	{attribute 'c++_compatible'}
	{attribute 'external_name' := 'FB_VN_ReadRegister_UDINT_GUID_B1D0CDA5_1E02_2B99_6D2D_309CAE674913'}
	{attribute 'TcIecLibraryType'}
	(* This FB reads a DINT register from the camera. Requires an open control channel (e.g. by calling FB_VN_GevCameraControl.OpenCamera() before) *)
	FUNCTION_BLOCK FB_VN_ReadRegister_UDINT
	VAR_INPUT
		(* The address of the register that should be read *)
		 {attribute 'GUID' := 'E1ED2436-3512-43FA-B927-3F71DEDDA853'}
		nAddress : GVCP_REGISTER_ADDRESS;
		(* OPTIONAL: The endianness of the register. 0 = Big, 1 = Little. Default: 0 *)
		nEndian : UINT;
		(* Reading the register is triggered by a rising edge at this input. *)
		bRead : BOOL;
	END_VAR
	VAR
		 {attribute 'hide'}
		_reserved1 : USINT;
	END_VAR
	VAR_INPUT
		(* Indicates the time before the function is cancelled. *)
		nTimeout : TIME := VISION_ADS_TIMEOUT;
	END_VAR
	VAR_OUTPUT
		(* The read value *)
		nValue : UDINT;
		(* This output remains TRUE until the function block has executed a command, but at the longest for the duration supplied to the 'nTimeout' input. While bBusy = TRUE, no new command will be accepted at the inputs. *)
		bBusy : BOOL;
		(* This output is switched to TRUE as soon as an error occurs during the execution of a command. The command-specific error code is contained in ‘nErrorId’. If the function block has a timeout error, 'bError' is TRUE and 'nErrorId' is 1861 (hexadecimal 0x745). Is reset to FALSE by the execution of a command at the inputs. *)
		bError : BOOL;
	END_VAR
	VAR
		 {attribute 'hide'}
		_reserved2 : UINT;
	END_VAR
	VAR_OUTPUT
		(* Contains the ADS error code or the command-specific error code of the last executed command. Is reset to 0 by the execution of a command at the inputs. *)
		nErrorId : UDINT;
	END_VAR
	VAR
		(* Internal reference to the corresponding TcVnGevImageProvider TcCOM module ID, which needs to be set via TC init symbol. *)
		{attribute 'TcInitSymbol'}
		{attribute 'TcCategoryOID' := 'TcVnGevImageProvider'}
		 {attribute 'GUID' := '18071995-0000-0000-0000-00000000000F'}
		oidITcVnGevImageProvider : OTCID;
		 {attribute 'hide'}
		_reserved3 : UINT_0_32;
		(* Internal reference to the corresponding TcVnGevImageProvider module. *)
		{attribute 'hide'}
		 {attribute 'GUID' := 'ED7659DB-95DC-4A4A-B62F-02C9870D5E81'}
		ipGevImageProvider : ITcVnGevImageProvider;
		(* Internal timestamp for timeout detection *)
		{attribute 'hide'}
		nTimeElapsed : TIME;
		(* Internal flag for rising edge detection *)
		{attribute 'hide'}
		bLastRead : BOOL;
		 {attribute 'hide'}
		_reserved4 : ARRAY [1..3] OF USINT;
	END_VAR


	(* Internal method *)
	{attribute 'hide'}
	METHOD FB_exit : BOOL
	VAR_INPUT
		(*  if TRUE, the exit method is called for exiting an instance that is copied afterwards (online change). *)
		bInCopyCode : BOOL;
	END_VAR
END_METHOD


	(* Internal method *)
	{attribute 'hide'}
	METHOD FB_init : BOOL
	VAR_INPUT
		(*  if TRUE, the retain variables are initialized (warm start / cold start) *)
		bInitRetains : BOOL;
		(*  if TRUE, the instance afterwards gets moved into the copy code (online change) *)
		bInCopyCode : BOOL;
	END_VAR
END_METHOD

END_FUNCTION_BLOCK

// Function Blocks/Camera Register Access/FB_VN_WriteRegister_UDINT

	{attribute 'c++_compatible'}
	{attribute 'external_name' := 'FB_VN_WriteRegister_UDINT_GUID_AF8CFF3D_C541_213B_73EF_5E560CA3A7B1'}
	{attribute 'TcIecLibraryType'}
	(* This FB writes a DINT value into a register on the camera. Requires an open control channel (e.g. by calling FB_VN_GevCameraControl.OpenCamera() before) *)
	FUNCTION_BLOCK FB_VN_WriteRegister_UDINT
	VAR_INPUT
		(* The address of the register that should be written *)
		 {attribute 'GUID' := 'E1ED2436-3512-43FA-B927-3F71DEDDA853'}
		nAddress : GVCP_REGISTER_ADDRESS;
		(* The value to write *)
		nValue : UDINT;
		(* OPTIONAL: The endianness of the register. 0 = Big, 1 = Little. Default: 0 *)
		nEndian : UINT;
		(* Writing the register is triggered by a rising edge at this input. *)
		bWrite : BOOL;
	END_VAR
	VAR
		 {attribute 'hide'}
		_reserved1 : USINT;
	END_VAR
	VAR_INPUT
		(* Indicates the time before the function is cancelled. *)
		nTimeout : TIME := VISION_ADS_TIMEOUT;
	END_VAR
	VAR_OUTPUT
		(* This output remains TRUE until the function block has executed a command, but at the longest for the duration supplied to the 'nTimeout' input. While bBusy = TRUE, no new command will be accepted at the inputs. *)
		bBusy : BOOL;
		(* This output is switched to TRUE as soon as an error occurs during the execution of a command. The command-specific error code is contained in ‘nErrorId’. If the function block has a timeout error, 'bError' is TRUE and 'nErrorId' is 1861 (hexadecimal 0x745). Is reset to FALSE by the execution of a command at the inputs. *)
		bError : BOOL;
	END_VAR
	VAR
		 {attribute 'hide'}
		_reserved2 : UINT;
	END_VAR
	VAR_OUTPUT
		(* Contains the ADS error code or the command-specific error code of the last executed command. Is reset to 0 by the execution of a command at the inputs. *)
		nErrorId : UDINT;
	END_VAR
	VAR
		(* Internal reference to the corresponding TcVnGevImageProvider TcCOM module ID, which needs to be set via TC init symbol. *)
		{attribute 'TcInitSymbol'}
		{attribute 'TcCategoryOID' := 'TcVnGevImageProvider'}
		 {attribute 'GUID' := '18071995-0000-0000-0000-00000000000F'}
		oidITcVnGevImageProvider : OTCID;
		 {attribute 'hide'}
		_reserved3 : UINT_0_32;
		(* Internal reference to the corresponding TcVnGevImageProvider module. *)
		{attribute 'hide'}
		 {attribute 'GUID' := 'ED7659DB-95DC-4A4A-B62F-02C9870D5E81'}
		ipGevImageProvider : ITcVnGevImageProvider;
		(* Internal timestamp for timeout detection *)
		{attribute 'hide'}
		nTimeElapsed : TIME;
		(* Internal flag for rising edge detection *)
		{attribute 'hide'}
		bLastWrite : BOOL;
		 {attribute 'hide'}
		_reserved4 : ARRAY [1..3] OF USINT;
	END_VAR


	(* Internal method *)
	{attribute 'hide'}
	METHOD FB_exit : BOOL
	VAR_INPUT
		(*  if TRUE, the exit method is called for exiting an instance that is copied afterwards (online change). *)
		bInCopyCode : BOOL;
	END_VAR
END_METHOD


	(* Internal method *)
	{attribute 'hide'}
	METHOD FB_init : BOOL
	VAR_INPUT
		(*  if TRUE, the retain variables are initialized (warm start / cold start) *)
		bInitRetains : BOOL;
		(*  if TRUE, the instance afterwards gets moved into the copy code (online change) *)
		bInCopyCode : BOOL;
	END_VAR
END_METHOD

END_FUNCTION_BLOCK

// Function Blocks/Camera Register Access/FB_VN_ReadRegister_ULINT

	{attribute 'c++_compatible'}
	{attribute 'external_name' := 'FB_VN_ReadRegister_ULINT_GUID_6D8277AF_24E6_2571_66A8_DA51E0B530F6'}
	{attribute 'TcIecLibraryType'}
	(* This FB reads a ULINT register from the camera. Requires an open control channel (e.g. by calling FB_VN_GevCameraControl.OpenCamera() before) *)
	FUNCTION_BLOCK FB_VN_ReadRegister_ULINT
	VAR_INPUT
		(* The address of the register that should be read *)
		 {attribute 'GUID' := 'E1ED2436-3512-43FA-B927-3F71DEDDA853'}
		nAddress : GVCP_REGISTER_ADDRESS;
		(* OPTIONAL: The endianness of the register. 0 = Big, 1 = Little. Default: 0 *)
		nEndian : UINT;
		(* Reading the register is triggered by a rising edge at this input. *)
		bRead : BOOL;
	END_VAR
	VAR
		 {attribute 'hide'}
		_reserved1 : USINT;
	END_VAR
	VAR_INPUT
		(* Indicates the time before the function is cancelled. *)
		nTimeout : TIME := VISION_ADS_TIMEOUT;
	END_VAR
	VAR
		 {attribute 'hide'}
		_reserved2 : UINT_0_32;
	END_VAR
	VAR_OUTPUT
		(* The read value *)
		nValue : ULINT;
		(* This output remains TRUE until the function block has executed a command, but at the longest for the duration supplied to the 'nTimeout' input. While bBusy = TRUE, no new command will be accepted at the inputs. *)
		bBusy : BOOL;
		(* This output is switched to TRUE as soon as an error occurs during the execution of a command. The command-specific error code is contained in ‘nErrorId’. If the function block has a timeout error, 'bError' is TRUE and 'nErrorId' is 1861 (hexadecimal 0x745). Is reset to FALSE by the execution of a command at the inputs. *)
		bError : BOOL;
	END_VAR
	VAR
		 {attribute 'hide'}
		_reserved3 : UINT;
	END_VAR
	VAR_OUTPUT
		(* Contains the ADS error code or the command-specific error code of the last executed command. Is reset to 0 by the execution of a command at the inputs. *)
		nErrorId : UDINT;
	END_VAR
	VAR
		(* Internal reference to the corresponding TcVnGevImageProvider TcCOM module ID, which needs to be set via TC init symbol. *)
		{attribute 'TcInitSymbol'}
		{attribute 'TcCategoryOID' := 'TcVnGevImageProvider'}
		 {attribute 'GUID' := '18071995-0000-0000-0000-00000000000F'}
		oidITcVnGevImageProvider : OTCID;
		 {attribute 'hide'}
		_reserved4 : UINT_0_32;
		(* Internal reference to the corresponding TcVnGevImageProvider module. *)
		{attribute 'hide'}
		 {attribute 'GUID' := 'ED7659DB-95DC-4A4A-B62F-02C9870D5E81'}
		ipGevImageProvider : ITcVnGevImageProvider;
		(* Internal timestamp for timeout detection *)
		{attribute 'hide'}
		nTimeElapsed : TIME;
		(* Internal flag for rising edge detection *)
		{attribute 'hide'}
		bLastRead : BOOL;
		 {attribute 'hide'}
		_reserved5 : ARRAY [1..3] OF USINT;
	END_VAR


	(* Internal method *)
	{attribute 'hide'}
	METHOD FB_exit : BOOL
	VAR_INPUT
		(*  if TRUE, the exit method is called for exiting an instance that is copied afterwards (online change). *)
		bInCopyCode : BOOL;
	END_VAR
END_METHOD


	(* Internal method *)
	{attribute 'hide'}
	METHOD FB_init : BOOL
	VAR_INPUT
		(*  if TRUE, the retain variables are initialized (warm start / cold start) *)
		bInitRetains : BOOL;
		(*  if TRUE, the instance afterwards gets moved into the copy code (online change) *)
		bInCopyCode : BOOL;
	END_VAR
END_METHOD

END_FUNCTION_BLOCK

// Function Blocks/Camera Register Access/FB_VN_WriteRegister_ULINT

	{attribute 'c++_compatible'}
	{attribute 'external_name' := 'FB_VN_WriteRegister_ULINT_GUID_F5D47CB9_E51C_2962_4F84_AA60BB261FC0'}
	{attribute 'TcIecLibraryType'}
	(* This FB writes a ULINT value into a register on the camera. Requires an open control channel (e.g. by calling FB_VN_GevCameraControl.OpenCamera() before) *)
	FUNCTION_BLOCK FB_VN_WriteRegister_ULINT
	VAR_INPUT
		(* The address of the register that should be written *)
		 {attribute 'GUID' := 'E1ED2436-3512-43FA-B927-3F71DEDDA853'}
		nAddress : GVCP_REGISTER_ADDRESS;
	END_VAR
	VAR
		 {attribute 'hide'}
		_reserved1 : UINT_0_32;
	END_VAR
	VAR_INPUT
		(* The value to write *)
		nValue : ULINT;
		(* OPTIONAL: The endianness of the register. 0 = Big, 1 = Little. Default: 0 *)
		nEndian : UINT;
		(* Writing the register is triggered by a rising edge at this input. *)
		bWrite : BOOL;
	END_VAR
	VAR
		 {attribute 'hide'}
		_reserved2 : USINT;
	END_VAR
	VAR_INPUT
		(* Indicates the time before the function is cancelled. *)
		nTimeout : TIME := VISION_ADS_TIMEOUT;
	END_VAR
	VAR_OUTPUT
		(* This output remains TRUE until the function block has executed a command, but at the longest for the duration supplied to the 'nTimeout' input. While bBusy = TRUE, no new command will be accepted at the inputs. *)
		bBusy : BOOL;
		(* This output is switched to TRUE as soon as an error occurs during the execution of a command. The command-specific error code is contained in ‘nErrorId’. If the function block has a timeout error, 'bError' is TRUE and 'nErrorId' is 1861 (hexadecimal 0x745). Is reset to FALSE by the execution of a command at the inputs. *)
		bError : BOOL;
	END_VAR
	VAR
		 {attribute 'hide'}
		_reserved3 : UINT;
	END_VAR
	VAR_OUTPUT
		(* Contains the ADS error code or the command-specific error code of the last executed command. Is reset to 0 by the execution of a command at the inputs. *)
		nErrorId : UDINT;
	END_VAR
	VAR
		(* Internal reference to the corresponding TcVnGevImageProvider TcCOM module ID, which needs to be set via TC init symbol. *)
		{attribute 'TcInitSymbol'}
		{attribute 'TcCategoryOID' := 'TcVnGevImageProvider'}
		 {attribute 'GUID' := '18071995-0000-0000-0000-00000000000F'}
		oidITcVnGevImageProvider : OTCID;
		 {attribute 'hide'}
		_reserved4 : UINT_0_32;
		(* Internal reference to the corresponding TcVnGevImageProvider module. *)
		{attribute 'hide'}
		 {attribute 'GUID' := 'ED7659DB-95DC-4A4A-B62F-02C9870D5E81'}
		ipGevImageProvider : ITcVnGevImageProvider;
		(* Internal timestamp for timeout detection *)
		{attribute 'hide'}
		nTimeElapsed : TIME;
		(* Internal flag for rising edge detection *)
		{attribute 'hide'}
		bLastWrite : BOOL;
		 {attribute 'hide'}
		_reserved5 : ARRAY [1..3] OF USINT;
	END_VAR


	(* Internal method *)
	{attribute 'hide'}
	METHOD FB_exit : BOOL
	VAR_INPUT
		(*  if TRUE, the exit method is called for exiting an instance that is copied afterwards (online change). *)
		bInCopyCode : BOOL;
	END_VAR
END_METHOD


	(* Internal method *)
	{attribute 'hide'}
	METHOD FB_init : BOOL
	VAR_INPUT
		(*  if TRUE, the retain variables are initialized (warm start / cold start) *)
		bInitRetains : BOOL;
		(*  if TRUE, the instance afterwards gets moved into the copy code (online change) *)
		bInCopyCode : BOOL;
	END_VAR
END_METHOD

END_FUNCTION_BLOCK

// Function Blocks/Camera Register Access/FB_VN_ReadMemory

	{attribute 'c++_compatible'}
	{attribute 'external_name' := 'FB_VN_ReadMemory_GUID_9CA954A7_F2A2_273A_543E_66E465761E40'}
	{attribute 'TcIecLibraryType'}
	(* This FB reads consecutive memory locations from the camera. Requires an open control channel (e.g. by calling FB_VN_GevCameraControl.OpenCamera() before) *)
	FUNCTION_BLOCK FB_VN_ReadMemory
	VAR_INPUT
		(* The address of the first byte to read from the camera (must be 32-bit aligned) *)
		 {attribute 'GUID' := 'E1ED2436-3512-43FA-B927-3F71DEDDA853'}
		nAddress : GVCP_REGISTER_ADDRESS;
		(* The number of bytes to read, starting with nAddress (must be a multiple of 4, not more than 536) *)
		nLength : UINT;
	END_VAR
	VAR
		 {attribute 'hide'}
		_reserved1 : UINT;
	END_VAR
	VAR_INPUT
		(* Pointer to the buffer where the read memory content is written to (The buffer must have a size of at least nLength bytes!) *)
		 {attribute 'GUID' := '18071995-0000-0000-0000-000000000018'}
		pBuffer : PVOID;
		(* Reading the memory is triggered by a rising edge at this input. *)
		bRead : BOOL;
	END_VAR
	VAR
		 {attribute 'hide'}
		_reserved2 : ARRAY [1..3] OF USINT;
	END_VAR
	VAR_INPUT
		(* Indicates the time before the function is cancelled. *)
		nTimeout : TIME := VISION_ADS_TIMEOUT;
	END_VAR
	VAR_OUTPUT
		(* This output remains TRUE until the function block has executed a command, but at the longest for the duration supplied to the 'nTimeout' input. While bBusy = TRUE, no new command will be accepted at the inputs. *)
		bBusy : BOOL;
		(* This output is switched to TRUE as soon as an error occurs during the execution of a command. The command-specific error code is contained in ‘nErrorId’. If the function block has a timeout error, 'bError' is TRUE and 'nErrorId' is 1861 (hexadecimal 0x745). Is reset to FALSE by the execution of a command at the inputs. *)
		bError : BOOL;
	END_VAR
	VAR
		 {attribute 'hide'}
		_reserved3 : UINT;
	END_VAR
	VAR_OUTPUT
		(* Contains the ADS error code or the command-specific error code of the last executed command. Is reset to 0 by the execution of a command at the inputs. *)
		nErrorId : UDINT;
	END_VAR
	VAR
		(* Internal reference to the corresponding TcVnGevImageProvider TcCOM module ID, which needs to be set via TC init symbol. *)
		{attribute 'TcInitSymbol'}
		{attribute 'TcCategoryOID' := 'TcVnGevImageProvider'}
		 {attribute 'GUID' := '18071995-0000-0000-0000-00000000000F'}
		oidITcVnGevImageProvider : OTCID;
		 {attribute 'hide'}
		_reserved4 : UINT_0_32;
		(* Internal reference to the corresponding TcVnGevImageProvider module. *)
		{attribute 'hide'}
		 {attribute 'GUID' := 'ED7659DB-95DC-4A4A-B62F-02C9870D5E81'}
		ipGevImageProvider : ITcVnGevImageProvider;
		(* Internal timestamp for timeout detection *)
		{attribute 'hide'}
		nTimeElapsed : TIME;
		(* Internal flag for rising edge detection *)
		{attribute 'hide'}
		bLastRead : BOOL;
		 {attribute 'hide'}
		_reserved5 : ARRAY [1..3] OF USINT;
	END_VAR


	(* Internal method *)
	{attribute 'hide'}
	METHOD FB_exit : BOOL
	VAR_INPUT
		(* If TRUE, the exit method is called for exiting an instance that is copied afterwards (online change). *)
		bInCopyCode : BOOL;
	END_VAR
END_METHOD


	(* Internal method *)
	{attribute 'hide'}
	METHOD FB_init : BOOL
	VAR_INPUT
		(* If TRUE, the retain variables are initialized (warm start / cold start) *)
		bInitRetains : BOOL;
		(* If TRUE, the instance afterwards gets moved into the copy code (online change) *)
		bInCopyCode : BOOL;
	END_VAR
END_METHOD

END_FUNCTION_BLOCK

// Function Blocks/Camera Register Access/FB_VN_WriteMemory

	{attribute 'c++_compatible'}
	{attribute 'external_name' := 'FB_VN_WriteMemory_GUID_898946BD_BBBB_2C1E_47B5_AFDF2B329C15'}
	{attribute 'TcIecLibraryType'}
	(* This FB writes data to consecutive memory locations on the camera. Requires an open control channel (e.g. by calling FB_VN_GevCameraControl.OpenCamera() before) *)
	FUNCTION_BLOCK FB_VN_WriteMemory
	VAR_INPUT
		(* The address of the first byte to write to the camera (must be 32-bit aligned) *)
		 {attribute 'GUID' := 'E1ED2436-3512-43FA-B927-3F71DEDDA853'}
		nAddress : GVCP_REGISTER_ADDRESS;
		(* The number of bytes to write, starting at nAddress (must be a multiple of 4, not more than 536) *)
		nLength : UINT;
	END_VAR
	VAR
		 {attribute 'hide'}
		_reserved1 : UINT;
	END_VAR
	VAR_INPUT
		(* Pointer to the data that should be written to the camera (must have a size of at least nLength bytes!) *)
		 {attribute 'GUID' := '18071995-0000-0000-0000-000000000018'}
		pData : PVOID;
		(* Writing the memory is triggered by a rising edge at this input. *)
		bWrite : BOOL;
	END_VAR
	VAR
		 {attribute 'hide'}
		_reserved2 : ARRAY [1..3] OF USINT;
	END_VAR
	VAR_INPUT
		(* Indicates the time before the function is cancelled. *)
		nTimeout : TIME := VISION_ADS_TIMEOUT;
	END_VAR
	VAR_OUTPUT
		(* This output remains TRUE until the function block has executed a command, but at the longest for the duration supplied to the 'nTimeout' input. While bBusy = TRUE, no new command will be accepted at the inputs. *)
		bBusy : BOOL;
		(* This output is switched to TRUE as soon as an error occurs during the execution of a command. The command-specific error code is contained in ‘nErrorId’. If the function block has a timeout error, 'bError' is TRUE and 'nErrorId' is 1861 (hexadecimal 0x745). Is reset to FALSE by the execution of a command at the inputs. *)
		bError : BOOL;
	END_VAR
	VAR
		 {attribute 'hide'}
		_reserved3 : UINT;
	END_VAR
	VAR_OUTPUT
		(* Contains the ADS error code or the command-specific error code of the last executed command. Is reset to 0 by the execution of a command at the inputs. *)
		nErrorId : UDINT;
		(* The number of bytes that have been successfully written to the camera. *)
		nBytesWritten : UINT;
	END_VAR
	VAR
		 {attribute 'hide'}
		_reserved4 : UINT;
		(* Internal reference to the corresponding TcVnGevImageProvider TcCOM module ID, which needs to be set via TC init symbol. *)
		{attribute 'TcInitSymbol'}
		{attribute 'TcCategoryOID' := 'TcVnGevImageProvider'}
		 {attribute 'GUID' := '18071995-0000-0000-0000-00000000000F'}
		oidITcVnGevImageProvider : OTCID;
		(* Internal reference to the corresponding TcVnGevImageProvider module. *)
		{attribute 'hide'}
		 {attribute 'GUID' := 'ED7659DB-95DC-4A4A-B62F-02C9870D5E81'}
		ipGevImageProvider : ITcVnGevImageProvider;
		(* Internal timestamp for timeout detection *)
		{attribute 'hide'}
		nTimeElapsed : TIME;
		(* Internal flag for rising edge detection *)
		{attribute 'hide'}
		bLastRead : BOOL;
		 {attribute 'hide'}
		_reserved5 : ARRAY [1..3] OF USINT;
	END_VAR


	(* Internal method *)
	{attribute 'hide'}
	METHOD FB_exit : BOOL
	VAR_INPUT
		(* If TRUE, the exit method is called for exiting an instance that is copied afterwards (online change). *)
		bInCopyCode : BOOL;
	END_VAR
END_METHOD


	(* Internal method *)
	{attribute 'hide'}
	METHOD FB_init : BOOL
	VAR_INPUT
		(* If TRUE, the retain variables are initialized (warm start / cold start) *)
		bInitRetains : BOOL;
		(* If TRUE, the instance afterwards gets moved into the copy code (online change) *)
		bInCopyCode : BOOL;
	END_VAR
END_METHOD

END_FUNCTION_BLOCK

// Function Blocks/Camera Register Access/FB_VN_ReadRegister_REAL

	{attribute 'c++_compatible'}
	{attribute 'external_name' := 'FB_VN_ReadRegister_REAL_GUID_EB9375A9_7535_2856_5B60_6EDD0CE066B0'}
	{attribute 'TcIecLibraryType'}
	(* This FB reads a REAL register from the camera. Requires an open control channel (e.g. by calling FB_VN_GevCameraControl.OpenCamera() before) *)
	FUNCTION_BLOCK FB_VN_ReadRegister_REAL
	VAR_INPUT
		(* The address of the register that should be read *)
		 {attribute 'GUID' := 'E1ED2436-3512-43FA-B927-3F71DEDDA853'}
		nAddress : GVCP_REGISTER_ADDRESS;
		(* OPTIONAL: The endianness of the register. 0 = Big, 1 = Little. Default: 0 *)
		nEndian : UINT;
		(* Reading the register is triggered by a rising edge at this input. *)
		bRead : BOOL;
	END_VAR
	VAR
		 {attribute 'hide'}
		_reserved1 : USINT;
	END_VAR
	VAR_INPUT
		(* Indicates the time before the function is cancelled. *)
		nTimeout : TIME := VISION_ADS_TIMEOUT;
	END_VAR
	VAR_OUTPUT
		(* The read value *)
		fValue : REAL;
		(* This output remains TRUE until the function block has executed a command, but at the longest for the duration supplied to the 'nTimeout' input. While bBusy = TRUE, no new command will be accepted at the inputs. *)
		bBusy : BOOL;
		(* This output is switched to TRUE as soon as an error occurs during the execution of a command. The command-specific error code is contained in ‘nErrorId’. If the function block has a timeout error, 'bError' is TRUE and 'nErrorId' is 1861 (hexadecimal 0x745). Is reset to FALSE by the execution of a command at the inputs. *)
		bError : BOOL;
	END_VAR
	VAR
		 {attribute 'hide'}
		_reserved2 : UINT;
	END_VAR
	VAR_OUTPUT
		(* Contains the ADS error code or the command-specific error code of the last executed command. Is reset to 0 by the execution of a command at the inputs. *)
		nErrorId : UDINT;
	END_VAR
	VAR
		(* Internal reference to the corresponding TcVnGevImageProvider TcCOM module ID, which needs to be set via TC init symbol. *)
		{attribute 'TcInitSymbol'}
		{attribute 'TcCategoryOID' := 'TcVnGevImageProvider'}
		 {attribute 'GUID' := '18071995-0000-0000-0000-00000000000F'}
		oidITcVnGevImageProvider : OTCID;
		 {attribute 'hide'}
		_reserved3 : UINT_0_32;
		(* Internal reference to the corresponding TcVnGevImageProvider module. *)
		{attribute 'hide'}
		 {attribute 'GUID' := 'ED7659DB-95DC-4A4A-B62F-02C9870D5E81'}
		ipGevImageProvider : ITcVnGevImageProvider;
		(* Internal timestamp for timeout detection *)
		{attribute 'hide'}
		nTimeElapsed : TIME;
		(* Internal flag for rising edge detection *)
		{attribute 'hide'}
		bLastRead : BOOL;
		 {attribute 'hide'}
		_reserved4 : ARRAY [1..3] OF USINT;
	END_VAR


	(* Internal method *)
	{attribute 'hide'}
	METHOD FB_exit : BOOL
	VAR_INPUT
		(*  if TRUE, the exit method is called for exiting an instance that is copied afterwards (online change). *)
		bInCopyCode : BOOL;
	END_VAR
END_METHOD


	(* Internal method *)
	{attribute 'hide'}
	METHOD FB_init : BOOL
	VAR_INPUT
		(*  if TRUE, the retain variables are initialized (warm start / cold start) *)
		bInitRetains : BOOL;
		(*  if TRUE, the instance afterwards gets moved into the copy code (online change) *)
		bInCopyCode : BOOL;
	END_VAR
END_METHOD

END_FUNCTION_BLOCK

// Function Blocks/Camera Register Access/FB_VN_WriteRegister_REAL

	{attribute 'c++_compatible'}
	{attribute 'external_name' := 'FB_VN_WriteRegister_REAL_GUID_FC95A1D0_F249_2125_5E8B_72E0441796A5'}
	{attribute 'TcIecLibraryType'}
	(* This FB writes a REAL value into a register on the camera. Requires an open control channel (e.g. by calling FB_VN_GevCameraControl.OpenCamera() before) *)
	FUNCTION_BLOCK FB_VN_WriteRegister_REAL
	VAR_INPUT
		(* The address of the register that should be written *)
		 {attribute 'GUID' := 'E1ED2436-3512-43FA-B927-3F71DEDDA853'}
		nAddress : GVCP_REGISTER_ADDRESS;
		(* The value to write *)
		fValue : REAL;
		(* OPTIONAL: The endianness of the register. 0 = Big, 1 = Little. Default: 0 *)
		nEndian : UINT;
		(* Writing the register is triggered by a rising edge at this input. *)
		bWrite : BOOL;
	END_VAR
	VAR
		 {attribute 'hide'}
		_reserved1 : USINT;
	END_VAR
	VAR_INPUT
		(* Indicates the time before the function is cancelled. *)
		nTimeout : TIME := VISION_ADS_TIMEOUT;
	END_VAR
	VAR_OUTPUT
		(* This output remains TRUE until the function block has executed a command, but at the longest for the duration supplied to the 'nTimeout' input. While bBusy = TRUE, no new command will be accepted at the inputs. *)
		bBusy : BOOL;
		(* This output is switched to TRUE as soon as an error occurs during the execution of a command. The command-specific error code is contained in ‘nErrorId’. If the function block has a timeout error, 'bError' is TRUE and 'nErrorId' is 1861 (hexadecimal 0x745). Is reset to FALSE by the execution of a command at the inputs. *)
		bError : BOOL;
	END_VAR
	VAR
		 {attribute 'hide'}
		_reserved2 : UINT;
	END_VAR
	VAR_OUTPUT
		(* Contains the ADS error code or the command-specific error code of the last executed command. Is reset to 0 by the execution of a command at the inputs. *)
		nErrorId : UDINT;
	END_VAR
	VAR
		(* Internal reference to the corresponding TcVnGevImageProvider TcCOM module ID, which needs to be set via TC init symbol. *)
		{attribute 'TcInitSymbol'}
		{attribute 'TcCategoryOID' := 'TcVnGevImageProvider'}
		 {attribute 'GUID' := '18071995-0000-0000-0000-00000000000F'}
		oidITcVnGevImageProvider : OTCID;
		 {attribute 'hide'}
		_reserved3 : UINT_0_32;
		(* Internal reference to the corresponding TcVnGevImageProvider module. *)
		{attribute 'hide'}
		 {attribute 'GUID' := 'ED7659DB-95DC-4A4A-B62F-02C9870D5E81'}
		ipGevImageProvider : ITcVnGevImageProvider;
		(* Internal timestamp for timeout detection *)
		{attribute 'hide'}
		nTimeElapsed : TIME;
		(* Internal flag for rising edge detection *)
		{attribute 'hide'}
		bLastWrite : BOOL;
		 {attribute 'hide'}
		_reserved4 : ARRAY [1..3] OF USINT;
	END_VAR


	(* Internal method *)
	{attribute 'hide'}
	METHOD FB_exit : BOOL
	VAR_INPUT
		(*  if TRUE, the exit method is called for exiting an instance that is copied afterwards (online change). *)
		bInCopyCode : BOOL;
	END_VAR
END_METHOD


	(* Internal method *)
	{attribute 'hide'}
	METHOD FB_init : BOOL
	VAR_INPUT
		(*  if TRUE, the retain variables are initialized (warm start / cold start) *)
		bInitRetains : BOOL;
		(*  if TRUE, the instance afterwards gets moved into the copy code (online change) *)
		bInCopyCode : BOOL;
	END_VAR
END_METHOD

END_FUNCTION_BLOCK

// Function Blocks/Image Processing/FB_VN_GeneralizedHoughBallard

	{attribute 'c++_compatible'}
	{attribute 'external_name' := 'FB_VN_GeneralizedHoughBallard_GUID_C8D436D3_9D4F_2963_727D_2C26455571C8'}
	{attribute 'TcIecLibraryType'}
	{attribute 'no_explicit_call' :='do not call this POU directly'}
	(* This FB provides the Generalized Hough Ballard functionality. First, set the parameters via the corresponding methods (optional, defaults are used otherwise). Then, set the template (required). Afterwards, the Detect method can be executed. *)
	FUNCTION_BLOCK FB_VN_GeneralizedHoughBallard
	VAR
		(* Internal stuff *)
		{attribute 'hide'}
		 {attribute 'GUID' := '18071995-0000-0000-0000-000000000018'}
		internal1 : PVOID;
		(* Internal stuff *)
		{attribute 'hide'}
		 {attribute 'GUID' := '18071995-0000-0000-0000-000000000018'}
		internal2 : PVOID;
		(* Internal stuff *)
		{attribute 'hide'}
		internal3 : BOOL;
		 {attribute 'hide'}
		_reserved1 : UINT_24_56;
	END_VAR


	(* Internal method *)
	{attribute 'hide'}
	METHOD FB_exit : BOOL
	VAR_INPUT
		(* if TRUE, the exit method is called for exiting an instance that is copied afterwards (online change). *)
		bInCopyCode : BOOL;
	END_VAR
END_METHOD


	(* Internal method *)
	{attribute 'hide'}
	METHOD FB_init : BOOL
	VAR_INPUT
		(* if TRUE, the retain variables are initialized (warm start / cold start) *)
		bInitRetains : BOOL;
		(* if TRUE, the instance afterwards gets moved into the copy code (online change) *)
		bInCopyCode : BOOL;
	END_VAR
END_METHOD


	(* Detect the template in an image (SetTemplate must have been called before). *)
	METHOD Detect : HRESULT
	VAR_INPUT
		(* Source image (1 channel, USINT) *)
 {attribute 'GUID' := '70D42C6D-6F4E-4719-8B29-2883D5D59B1C'}
				ipImage : ITcVnImage;
		(* Returns the centers of the detected template positions (ContainerType_Vector_TcVnPoint2_REAL; Non-zero interface pointers are reused.) *)
 {attribute 'GUID' := 'BC72B333-E095-465B-9693-7979773CA3B8'}
				ipPositions : REFERENCE TO ITcVnContainer;
	END_VAR
END_METHOD


	(* Sets the canny edge detection thresholds. *)
	METHOD SetCannyThreshold : HRESULT
	VAR_INPUT
		(* Low threshold (> 0) *)
		nLow : DINT;
		(* High threshold (> nLow, usually 2 to 3 * nLow) *)
		nHigh : DINT;
	END_VAR
END_METHOD


	(* Sets the inverted ratio of the accumulator size in relation to the source image's size (e.g. a value of 2 means that the size is halved in both directions.) *)
	METHOD SetInvAccuRatio : HRESULT
	VAR_INPUT
		(* Inverted accumulator ratio (> 0) *)
		fInvAccuRatio : LREAL;
	END_VAR
END_METHOD


	(* Sets the number of R-table levels. *)
	METHOD SetLevels : HRESULT
	VAR_INPUT
		(* Number of R-table levels (> 0) *)
		nLevels : DINT;
	END_VAR
END_METHOD


	(* Sets the minimum distance between the centers of different objects. *)
	METHOD SetMinDist : HRESULT
	VAR_INPUT
		(* Minimum distance (> 0) *)
		fMinDist : LREAL;
	END_VAR
END_METHOD


	(* Sets the template image to search for in the Detect method. *)
	METHOD SetTemplate : HRESULT
	VAR_INPUT
		(* Template image (1 channel, USINT) *)
 {attribute 'GUID' := '70D42C6D-6F4E-4719-8B29-2883D5D59B1C'}
				ipImage : ITcVnImage;
	END_VAR
END_METHOD


	(* Sets the accumulator threshold, i.e. the number of votes required to detect a match (too small values lead to false detections). *)
	METHOD SetVotesThreshold : HRESULT
	VAR_INPUT
		(* Number of votes required to detect a match (> 0) *)
		nVotes : DINT;
	END_VAR
END_METHOD

END_FUNCTION_BLOCK

// Function Blocks/Image Processing/FB_VN_SSIM

	{attribute 'c++_compatible'}
	{attribute 'external_name' := 'FB_VN_SSIM_GUID_28E6E97D_2E13_23A7_7751_F8A715064107'}
	{attribute 'TcIecLibraryType'}
	{attribute 'no_explicit_call' :='do not call this POU directly'}
	(* This FB provides the structural similarity (SSIM) functionality. First, set the reference image. Afterwards, the Compute method can be executed. *)
	FUNCTION_BLOCK FB_VN_SSIM
	VAR
		(* Internal stuff *)
		{attribute 'hide'}
		 {attribute 'GUID' := '18071995-0000-0000-0000-000000000018'}
		internal1 : PVOID;
	END_VAR


	(* Internal method *)
	{attribute 'hide'}
	METHOD FB_exit : BOOL
	VAR_INPUT
		(* if TRUE, the exit method is called for exiting an instance that is copied afterwards (online change). *)
		bInCopyCode : BOOL;
	END_VAR
END_METHOD


	(* Internal method *)
	{attribute 'hide'}
	METHOD FB_init : BOOL
	VAR_INPUT
		(* if TRUE, the retain variables are initialized (warm start / cold start) *)
		bInitRetains : BOOL;
		(* if TRUE, the instance afterwards gets moved into the copy code (online change) *)
		bInCopyCode : BOOL;
	END_VAR
END_METHOD


	(* Compute the structural similarity (SetReference must have been called before). *)
	METHOD Compute : HRESULT
	VAR_INPUT
		(* Source image (USINT) *)
 {attribute 'GUID' := '70D42C6D-6F4E-4719-8B29-2883D5D59B1C'}
				ipSrcImage : ITcVnImage;
		(* Returns the SSIM (REAL, values from 0 to 1) *)
 {attribute 'GUID' := '70D42C6D-6F4E-4719-8B29-2883D5D59B1C'}
				ipSSIM : REFERENCE TO ITcVnImage;
	END_VAR
END_METHOD


	(* Sets the reference image, used by the SSIM method. *)
	METHOD SetReference : HRESULT
	VAR_INPUT
		(* Reference image (USINT) *)
 {attribute 'GUID' := '70D42C6D-6F4E-4719-8B29-2883D5D59B1C'}
				ipImage : ITcVnImage;
	END_VAR
END_METHOD

END_FUNCTION_BLOCK

// Functions/Control Functions/F_VN_StartAbsWatchdog

	{attribute 'TcIecLibraryType'}
	{attribute 'external_name' := 'F_VN_StartAbsWatchdog_GUID_5DDC619B_43C5_2ACF_6EB3_2E2FDA2A7E7B'}
	(* Starts a cooperative watchdog given an absolute stop time. *)
	FUNCTION F_VN_StartAbsWatchdog : HRESULT
	VAR_INPUT
		tStop	:	DINT;	(* Stop time in us *)
		hrPrev	:	HRESULT;	(* HRESULT indicating the result of previous operations (If SUCCEEDED(hrPrev) equals false, no operation is executed.) *)
	END_VAR

END_FUNCTION

// Functions/Control Functions/F_VN_StartAbsWatchdogExp

	{attribute 'TcIecLibraryType'}
	{attribute 'external_name' := 'F_VN_StartAbsWatchdogExp_GUID_CD9691CE_048C_265B_4306_B079C89C1BAD'}
	(* Start a cooperative watchdog given an absolute stop time. (expert function) *)
	FUNCTION F_VN_StartAbsWatchdogExp : HRESULT
	VAR_INPUT
		tStop	:	DINT;	(* Stop time in us *)
		eWatchdogAccType	:	ETcWatchdogAccumulationType;	(* Accumalation method used for combining the results of multiple functions enclosed by this watchdog *)
		hrPrev	:	HRESULT;	(* HRESULT indicating the result of previous operations (If SUCCEEDED(hrPrev) equals false, no operation is executed.) *)
	END_VAR

END_FUNCTION

// Functions/Control Functions/F_VN_StartRelWatchdog

	{attribute 'TcIecLibraryType'}
	{attribute 'external_name' := 'F_VN_StartRelWatchdog_GUID_A65F7A02_71F5_249F_492A_6E1D109B5534'}
	(* Starts a cooperative watchdog given a stop time relative to the current time. *)
	FUNCTION F_VN_StartRelWatchdog : HRESULT
	VAR_INPUT
		tStop	:	DINT;	(* Stop time in us *)
		hrPrev	:	HRESULT;	(* HRESULT indicating the result of previous operations (If SUCCEEDED(hrPrev) equals false, no operation is executed.) *)
	END_VAR

END_FUNCTION

// Functions/Control Functions/F_VN_StartRelWatchdogExp

	{attribute 'TcIecLibraryType'}
	{attribute 'external_name' := 'F_VN_StartRelWatchdogExp_GUID_A51FB774_F353_2EAF_6C85_EA9615EA8D2D'}
	(* Start a cooperative watchdog given a stop time relative to the current time. (expert function) *)
	FUNCTION F_VN_StartRelWatchdogExp : HRESULT
	VAR_INPUT
		tStop	:	DINT;	(* Stop time in us *)
		eWatchdogAccType	:	ETcWatchdogAccumulationType;	(* Accumalation method used for combining the results of multiple functions enclosed by this watchdog *)
		hrPrev	:	HRESULT;	(* HRESULT indicating the result of previous operations (If SUCCEEDED(hrPrev) equals false, no operation is executed.) *)
	END_VAR

END_FUNCTION

// Functions/Control Functions/F_VN_StopWatchdog

	{attribute 'TcIecLibraryType'}
	{attribute 'external_name' := 'F_VN_StopWatchdog_GUID_CF8714D2_1F6E_252E_5569_FC7334C94EBE'}
	(* Stops a watchdog and provide runtime information. *)
	FUNCTION F_VN_StopWatchdog : HRESULT
	VAR_INPUT
		hrStartWatchdog	:	HRESULT;	(* HRESULT indicating the result of the function used to start the watchdog (If SUCCEEDED(hrStartWatchdog) equals false, no operation is executed.) *)
	END_VAR
	VAR_OUTPUT
		nFunctionsMonitored	:	ULINT;	(* Returns the number of functions monitored *)
		nFractionProcessed	:	UDINT;	(* Returns the fraction processed accumulated over the monitored functions in percent *)
		tRest	:	DINT;	(* Returns the remaining computation time in us (may be negative) *)
	END_VAR

END_FUNCTION

// Functions/Image Segmentation/F_VN_AdaptiveThreshold

	{attribute 'TcIecLibraryType'}
	{attribute 'external_name' := 'F_VN_AdaptiveThreshold_GUID_21D34C79_9416_2C03_5A79_D5C5829F2427'}
	(* Apply an adaptive threshold to a gray level image. *)
	FUNCTION F_VN_AdaptiveThreshold : HRESULT
	VAR_INPUT
		ipSrcImage	:	ITcVnImage;	(* Source image (1 channel, elements of type USINT) *)
		ipDestImage	:	REFERENCE TO ITcVnImage;	(* Destination image (An appropriate destination image will be created if required.) *)
		fMaxValue	:	LREAL;	(* Value assigned to pixels for which the threshold condition is true *)
		hrPrev	:	HRESULT;	(* HRESULT indicating the result of previous operations (If SUCCEEDED(hrPrev) equals false, no operation is executed.) *)
	END_VAR

END_FUNCTION

// Functions/Image Segmentation/F_VN_AdaptiveThresholdExp

	{attribute 'TcIecLibraryType'}
	{attribute 'external_name' := 'F_VN_AdaptiveThresholdExp_GUID_7471C955_6BFB_2805_5D4B_761FB5541703'}
	(* Apply an adaptive threshold to a gray level image. (expert function) *)
	FUNCTION F_VN_AdaptiveThresholdExp : HRESULT
	VAR_INPUT
		ipSrcImage	:	ITcVnImage;	(* Source image (1 channel, elements of type USINT) *)
		ipDestImage	:	REFERENCE TO ITcVnImage;	(* Destination image (An appropriate destination image will be created if required.) *)
		fMaxValue	:	LREAL;	(* Value assigned to pixels for which the threshold condition is true *)
		eAdaptiveMethod	:	ETcVnAdaptiveThresholdMethod;	(* Adaptive threshold method to be applied (MEAN: threshold value will be calculated as a mean of the nBlockSize x nBlockSize neighborhood of (x,y) minus fConstant. GAUSSIAN: threshold value is a weighted sum (cross-correlation with a Gaussian window) of the nBlockSize x nBlockSize neighborhood of (x,y) minus fConstant. *)
		eThresholdType	:	ETcVnThresholdType;	(* Threshold type to be applied (only BINARY and BINARY_INV are supported) *)
		nBlockSize	:	UDINT;	(* Size of the pixel neighborhood to calculate the local threshold (3, 5, 7, ...) *)
		fConstant	:	LREAL;	(* Constant that is subtracted from the weighted mean of the pixel neighborhood, which leads to the local threshold *)
		hrPrev	:	HRESULT;	(* HRESULT indicating the result of previous operations (If SUCCEEDED(hrPrev) equals false, no operation is executed.) *)
	END_VAR

END_FUNCTION

// Functions/Image Segmentation/F_VN_CheckColorRange

	{attribute 'TcIecLibraryType'}
	{attribute 'external_name' := 'F_VN_CheckColorRange_GUID_CF6AA11C_2FA1_26AE_495C_D33F4056756F'}
	(* Check if the pixel values of an image lie in a given range. The destination image has the same size as the source image but only one channel with
          a pixel element size of 8 bit. Its elements are set to 255 if the corresponding pixels of the source image are in the checked range and set to 0 otherwise. *)
	FUNCTION F_VN_CheckColorRange : HRESULT
	VAR_INPUT
		ipSrcImage	:	ITcVnImage;	(* Source image *)
		ipDestImage	:	REFERENCE TO ITcVnImage;	(* Destination image (An appropriate destination image will be created if required.) *)
	END_VAR
	VAR_IN_OUT
		aLowerBounds	:	TcVnVector4_LREAL;	(* Channel-wise lower bounds (Unused channels are ignored.) *)
		aUpperBounds	:	TcVnVector4_LREAL;	(* Channel-wise upper bounds (Unused channels are ignored.) *)
	END_VAR
	VAR_INPUT
		hrPrev	:	HRESULT;	(* HRESULT indicating the result of previous operations (If SUCCEEDED(hrPrev) equals false, no operation is executed.) *)
	END_VAR

END_FUNCTION

// Functions/Image Segmentation/F_VN_DoubleThreshold

	{attribute 'TcIecLibraryType'}
	{attribute 'external_name' := 'F_VN_DoubleThreshold_GUID_E8588BF8_9D31_20A1_4DC9_53355F6E668C'}
	(* Apply a double threshold (also called hysteresis threshold) using morphological reconstruction. *)
	FUNCTION F_VN_DoubleThreshold : HRESULT
	VAR_INPUT
		ipSrcImage	:	ITcVnImage;	(* Source image (USINT, UINT, INT, REAL, or LREAL, 1 channel) *)
		ipDestImage	:	REFERENCE TO ITcVnImage;	(* Destination image (An appropriate destination image will be created if required.) *)
		fLowThreshold	:	LREAL;	(* Low threshold determinining the shape of found regions *)
		fHighThreshold	:	LREAL;	(* High threshold selecting found regions (Each region must at least contain a single pixel if the high threshold is applied.) *)
		fMaxValue	:	LREAL;	(* Maximum pixel value *)
		hrPrev	:	HRESULT;	(* HRESULT indicating the result of previous operations (If SUCCEEDED(hrPrev) equals false, no operation is executed.) *)
	END_VAR

END_FUNCTION

// Functions/Image Segmentation/F_VN_SauvolaThreshold

	{attribute 'TcIecLibraryType'}
	{attribute 'external_name' := 'F_VN_SauvolaThreshold_GUID_EFF2D812_CB05_27C3_5A25_22EA14357C42'}
	(* Apply Sauvola local threshold to source image. *)
	FUNCTION F_VN_SauvolaThreshold : HRESULT
	VAR_INPUT
		ipSrcImage	:	ITcVnImage;	(* Source image (USINT, UINT, INT, REAL, or LREAL, 1 channel) *)
		pipDestImage	:	REFERENCE TO ITcVnImage;	(* Destination image (An appropriate single channel destination image will be created if required.)) *)
		nBlockSize	:	UDINT;	(* Size of the pixel neighborhood to calculate the local threshold (3, 5, 7, ...) *)
		fParamK	:	LREAL;	(* parameter K which takes positive values in range (0,1). Recommended are K in range [0.2, 0.5] *)
		fMaxSigma	:	LREAL;	(* Maximum value of the standard deviation, required to be strictly positive. (fMaxSigma = 128 for a grayscale document).   *)
		eThresholdType	:	ETcVnThresholdType;	(* Threshold type to be applied. Supported are TCVN_TT_BINARY and TCVN_TT_BINARY_INV. *)
		hrPrev	:	HRESULT;	(* HRESULT indicating the result of previous operations (If SUCCEEDED(hrPrev) equals false, no operation is executed.) *)
	END_VAR

END_FUNCTION

// Functions/Image Segmentation/F_VN_Threshold

	{attribute 'TcIecLibraryType'}
	{attribute 'external_name' := 'F_VN_Threshold_GUID_64D0BD16_75B3_27A3_6D7B_7895F16EABC2'}
	(* Apply a fixed threshold or a dynamic threshold according to Otsu. *)
	FUNCTION F_VN_Threshold : HRESULT
	VAR_INPUT
		ipSrcImage	:	ITcVnImage;	(* Source image (For Otsu and Triangle threshold types, only 1 channel of TCVN_ET_USINT is supported) *)
		ipDestImage	:	REFERENCE TO ITcVnImage;	(* Destination image (An appropriate destination image will be created if required.) *)
		fThreshold	:	LREAL;	(* Fixed threshold (unused if dynamic thresholding is selected) *)
		fMaxValue	:	LREAL;	(* Maximum pixel value *)
		eThresholdType	:	ETcVnThresholdType;	(* Threshold type to be applied *)
		hrPrev	:	HRESULT;	(* HRESULT indicating the result of previous operations (If SUCCEEDED(hrPrev) equals false, no operation is executed.) *)
	END_VAR

END_FUNCTION

// Functions/Image Segmentation/F_VN_WatershedSegmentationExp

	{attribute 'TcIecLibraryType'}
	{attribute 'external_name' := 'F_VN_WatershedSegmentationExp_GUID_952B7815_FB0A_2C88_63CD_95BD80B1A3F1'}
	(* Apply a marker-based watershed segmentation. (expert function) *)
	FUNCTION F_VN_WatershedSegmentationExp : HRESULT
	VAR_INPUT
		ipSrcImage	:	ITcVnImage;	(* Source image (USINT, 3 channels) *)
		ipDestImage	:	REFERENCE TO ITcVnImage;	(* Destination image (DINT, 1 channel. An appropriate image will be created if required.) *)
		ipMarkers	:	ITcVnImage;	(* Marker image (DINT, 1 channel) *)
		hrPrev	:	HRESULT;	(* HRESULT indicating the result of previous operations (If SUCCEEDED(hrPrev) equals false, no operation is executed.) *)
	END_VAR

END_FUNCTION

// Functions/Algebraic Container Operations/F_VN_AddContainers

	{attribute 'TcIecLibraryType'}
	{attribute 'external_name' := 'F_VN_AddContainers_GUID_A4A758D3_B693_270F_582C_436EA4E8894B'}
	(* Element-wise addition of two containers (same length and type). *)
	FUNCTION F_VN_AddContainers : HRESULT
	VAR_INPUT
		ipSrcContainer1	:	ITcVnContainer;	(* Source container 1 *)
		ipSrcContainer2	:	ITcVnContainer;	(* Source container 2 *)
		ipDestContainer	:	REFERENCE TO ITcVnContainer;	(* Returns the resulting container *)
		hrPrev	:	HRESULT;	(* HRESULT indicating the result of previous operations (If SUCCEEDED(hrPrev) equals false, no operation is executed.) *)
	END_VAR

END_FUNCTION

// Functions/Algebraic Container Operations/F_VN_BitwiseAndContainers

	{attribute 'TcIecLibraryType'}
	{attribute 'external_name' := 'F_VN_BitwiseAndContainers_GUID_7B1A4119_9033_27D1_4989_95CFF8F6A877'}
	(* Element-wise application of a bit-wise AND operator to two containers (same length and type, integer only). *)
	FUNCTION F_VN_BitwiseAndContainers : HRESULT
	VAR_INPUT
		ipSrcContainer1	:	ITcVnContainer;	(* Source container 1 *)
		ipSrcContainer2	:	ITcVnContainer;	(* Source container 2 *)
		ipDestContainer	:	REFERENCE TO ITcVnContainer;	(* Returns the resulting container *)
		hrPrev	:	HRESULT;	(* HRESULT indicating the result of previous operations (If SUCCEEDED(hrPrev) equals false, no operation is executed.) *)
	END_VAR

END_FUNCTION

// Functions/Algebraic Container Operations/F_VN_BitwiseNotContainer

	{attribute 'TcIecLibraryType'}
	{attribute 'external_name' := 'F_VN_BitwiseNotContainer_GUID_677B5AFD_5936_2FE2_4E5E_41D97D3F2556'}
	(* Element-wise application of a bit-wise NOT operator to a container (integer only). *)
	FUNCTION F_VN_BitwiseNotContainer : HRESULT
	VAR_INPUT
		ipSrcContainer	:	ITcVnContainer;	(* Source container *)
		ipDestContainer	:	REFERENCE TO ITcVnContainer;	(* Returns the resulting container *)
		hrPrev	:	HRESULT;	(* HRESULT indicating the result of previous operations (If SUCCEEDED(hrPrev) equals false, no operation is executed.) *)
	END_VAR

END_FUNCTION

// Functions/Algebraic Container Operations/F_VN_BitwiseOrContainers

	{attribute 'TcIecLibraryType'}
	{attribute 'external_name' := 'F_VN_BitwiseOrContainers_GUID_601CC025_F29A_2F65_5E34_7511FDC320A5'}
	(* Element-wise application of a bit-wise OR operator to two containers (same length and type, integer only). *)
	FUNCTION F_VN_BitwiseOrContainers : HRESULT
	VAR_INPUT
		ipSrcContainer1	:	ITcVnContainer;	(* Source container 1 *)
		ipSrcContainer2	:	ITcVnContainer;	(* Source container 2 *)
		ipDestContainer	:	REFERENCE TO ITcVnContainer;	(* Returns the resulting container *)
		hrPrev	:	HRESULT;	(* HRESULT indicating the result of previous operations (If SUCCEEDED(hrPrev) equals false, no operation is executed.) *)
	END_VAR

END_FUNCTION

// Functions/Algebraic Container Operations/F_VN_BitwiseXorContainers

	{attribute 'TcIecLibraryType'}
	{attribute 'external_name' := 'F_VN_BitwiseXorContainers_GUID_20653E44_9C4F_2AAB_4489_545C60B0E27D'}
	(* Element-wise application of a bit-wise XOR operator to two containers (same length and type, integer only). *)
	FUNCTION F_VN_BitwiseXorContainers : HRESULT
	VAR_INPUT
		ipSrcContainer1	:	ITcVnContainer;	(* Source container 1 *)
		ipSrcContainer2	:	ITcVnContainer;	(* Source container 2 *)
		ipDestContainer	:	REFERENCE TO ITcVnContainer;	(* Returns the resulting container *)
		hrPrev	:	HRESULT;	(* HRESULT indicating the result of previous operations (If SUCCEEDED(hrPrev) equals false, no operation is executed.) *)
	END_VAR

END_FUNCTION

// Functions/Algebraic Container Operations/F_VN_DivideContainers

	{attribute 'TcIecLibraryType'}
	{attribute 'external_name' := 'F_VN_DivideContainers_GUID_DF15C491_305F_25C3_5334_6E9E5C6BBB26'}
	(* Element-wise division of two containers (same length and type). In case of integer division by zero, the resulting element is set to 0 and S_DIVISION_BY_ZERO is returned instead of S_OK (value can be changed in F_VN_DivideContainersExp). *)
	FUNCTION F_VN_DivideContainers : HRESULT
	VAR_INPUT
		ipSrcContainer1	:	ITcVnContainer;	(* Source container 1 *)
		ipSrcContainer2	:	ITcVnContainer;	(* Source container 2 *)
		ipDestContainer	:	REFERENCE TO ITcVnContainer;	(* Returns the resulting container *)
		hrPrev	:	HRESULT;	(* HRESULT indicating the result of previous operations (If SUCCEEDED(hrPrev) equals false, no operation is executed.) *)
	END_VAR

END_FUNCTION

// Functions/Algebraic Container Operations/F_VN_DivideContainersExp

	{attribute 'TcIecLibraryType'}
	{attribute 'external_name' := 'F_VN_DivideContainersExp_GUID_C7080283_F2FC_2BE1_6B51_D2B17BA50E6B'}
	(* Element-wise division of two containers (same length and type). In case of integer division by zero, the resulting element is set to nIntDivideByZeroResult and S_DIVISION_BY_ZERO is returned instead of S_OK. (expert function) *)
	FUNCTION F_VN_DivideContainersExp : HRESULT
	VAR_INPUT
		ipSrcContainer1	:	ITcVnContainer;	(* Source container 1 *)
		ipSrcContainer2	:	ITcVnContainer;	(* Source container 2 *)
		ipDestContainer	:	REFERENCE TO ITcVnContainer;	(* Returns the resulting container *)
		nIntDivideByZeroResult	:	LINT;	(* Value set as result in case of integer division by zero *)
		hrPrev	:	HRESULT;	(* HRESULT indicating the result of previous operations (If SUCCEEDED(hrPrev) equals false, no operation is executed.) *)
	END_VAR

END_FUNCTION

// Functions/Algebraic Container Operations/F_VN_MaxContainer

	{attribute 'TcIecLibraryType'}
	{attribute 'external_name' := 'F_VN_MaxContainer_GUID_1788AA2E_2C0C_2988_522D_B821EA1FA28C'}
	(* Element-wise maximum of two containers (same length and type). *)
	FUNCTION F_VN_MaxContainer : HRESULT
	VAR_INPUT
		ipSrcContainer1	:	ITcVnContainer;	(* Source container 1 *)
		ipSrcContainer2	:	ITcVnContainer;	(* Source container 2 *)
		ipDestContainer	:	REFERENCE TO ITcVnContainer;	(* Returns the resulting container *)
		hrPrev	:	HRESULT;	(* HRESULT indicating the result of previous operations (If SUCCEEDED(hrPrev) equals false, no operation is executed.) *)
	END_VAR

END_FUNCTION

// Functions/Algebraic Container Operations/F_VN_MinContainer

	{attribute 'TcIecLibraryType'}
	{attribute 'external_name' := 'F_VN_MinContainer_GUID_9DE933AC_C9A4_2FE8_69EF_9330308B2CB8'}
	(* Element-wise minimum of two containers (same length and type). *)
	FUNCTION F_VN_MinContainer : HRESULT
	VAR_INPUT
		ipSrcContainer1	:	ITcVnContainer;	(* Source container 1 *)
		ipSrcContainer2	:	ITcVnContainer;	(* Source container 2 *)
		ipDestContainer	:	REFERENCE TO ITcVnContainer;	(* Returns the resulting container *)
		hrPrev	:	HRESULT;	(* HRESULT indicating the result of previous operations (If SUCCEEDED(hrPrev) equals false, no operation is executed.) *)
	END_VAR

END_FUNCTION

// Functions/Algebraic Container Operations/F_VN_MultiplyContainers

	{attribute 'TcIecLibraryType'}
	{attribute 'external_name' := 'F_VN_MultiplyContainers_GUID_85532C27_4C81_2B2C_5377_9AE5FB91991D'}
	(* Element-wise multiplication of two containers (same length and type). *)
	FUNCTION F_VN_MultiplyContainers : HRESULT
	VAR_INPUT
		ipSrcContainer1	:	ITcVnContainer;	(* Source container 1 *)
		ipSrcContainer2	:	ITcVnContainer;	(* Source container 2 *)
		ipDestContainer	:	REFERENCE TO ITcVnContainer;	(* Returns the resulting container *)
		hrPrev	:	HRESULT;	(* HRESULT indicating the result of previous operations (If SUCCEEDED(hrPrev) equals false, no operation is executed.) *)
	END_VAR

END_FUNCTION

// Functions/Algebraic Container Operations/F_VN_MultiplyWithContainerElements1

	{attribute 'TcIecLibraryType'}
	{attribute 'external_name' := 'F_VN_MultiplyWithContainerElements1_GUID_AA2C6728_58F5_2B7C_40EB_0D40566AE058'}
	(* Multiply each container element with a value. *)
	FUNCTION F_VN_MultiplyWithContainerElements1 : HRESULT
	VAR_INPUT
		fValue	:	LREAL;	(* Value *)
		ipContainer	:	ITcVnContainer;	(* Container with 1-dimensional elements *)
		hrPrev	:	HRESULT;	(* HRESULT indicating the result of previous operations (If SUCCEEDED(hrPrev) equals false, no operation is executed.) *)
	END_VAR

END_FUNCTION

// Functions/Algebraic Container Operations/F_VN_MultiplyWithContainerElements2

	{attribute 'TcIecLibraryType'}
	{attribute 'external_name' := 'F_VN_MultiplyWithContainerElements2_GUID_275EB9AF_C7C8_24C4_6042_96A1E9F755A5'}
	(* Multiply each container element with a value. *)
	FUNCTION F_VN_MultiplyWithContainerElements2 : HRESULT
	VAR_IN_OUT
		aValue	:	TcVnVector2_LREAL;	(* Value *)
	END_VAR
	VAR_INPUT
		ipContainer	:	ITcVnContainer;	(* Container with 2-dimensional elements *)
		hrPrev	:	HRESULT;	(* HRESULT indicating the result of previous operations (If SUCCEEDED(hrPrev) equals false, no operation is executed.) *)
	END_VAR

END_FUNCTION

// Functions/Algebraic Container Operations/F_VN_MultiplyWithContainerElements3

	{attribute 'TcIecLibraryType'}
	{attribute 'external_name' := 'F_VN_MultiplyWithContainerElements3_GUID_8C3901C4_61E8_2CF7_6C1A_D8838E998C58'}
	(* Multiply each container element with a value. *)
	FUNCTION F_VN_MultiplyWithContainerElements3 : HRESULT
	VAR_IN_OUT
		aValue	:	TcVnVector3_LREAL;	(* Value *)
	END_VAR
	VAR_INPUT
		ipContainer	:	ITcVnContainer;	(* Container with 3-dimensional elements *)
		hrPrev	:	HRESULT;	(* HRESULT indicating the result of previous operations (If SUCCEEDED(hrPrev) equals false, no operation is executed.) *)
	END_VAR

END_FUNCTION

// Functions/Algebraic Container Operations/F_VN_MultiplyWithContainerElements4

	{attribute 'TcIecLibraryType'}
	{attribute 'external_name' := 'F_VN_MultiplyWithContainerElements4_GUID_4DEA3EF0_9801_2473_6BCB_52084F6AF1B0'}
	(* Multiply each container element with a value. *)
	FUNCTION F_VN_MultiplyWithContainerElements4 : HRESULT
	VAR_IN_OUT
		aValue	:	TcVnVector4_LREAL;	(* Value *)
	END_VAR
	VAR_INPUT
		ipContainer	:	ITcVnContainer;	(* Container with 4-dimensional elements *)
		hrPrev	:	HRESULT;	(* HRESULT indicating the result of previous operations (If SUCCEEDED(hrPrev) equals false, no operation is executed.) *)
	END_VAR

END_FUNCTION

// Functions/Algebraic Container Operations/F_VN_NegateContainer

	{attribute 'TcIecLibraryType'}
	{attribute 'external_name' := 'F_VN_NegateContainer_GUID_978A07E4_251D_2054_42DD_18696042ED1B'}
	(* Element-wise negation of a container (two's complement). *)
	FUNCTION F_VN_NegateContainer : HRESULT
	VAR_INPUT
		ipSrcContainer	:	ITcVnContainer;	(* Source container *)
		ipDestContainer	:	REFERENCE TO ITcVnContainer;	(* Returns the resulting container (same type as ipSrcContainer) *)
		hrPrev	:	HRESULT;	(* HRESULT indicating the result of previous operations (If SUCCEEDED(hrPrev) equals false, no operation is executed.) *)
	END_VAR

END_FUNCTION

// Functions/Algebraic Container Operations/F_VN_SubtractContainers

	{attribute 'TcIecLibraryType'}
	{attribute 'external_name' := 'F_VN_SubtractContainers_GUID_BDC6CE7B_D22B_293B_5FB8_59DA77444152'}
	(* Element-wise subtraction of two containers (same length and type). *)
	FUNCTION F_VN_SubtractContainers : HRESULT
	VAR_INPUT
		ipSrcContainer1	:	ITcVnContainer;	(* Source container 1 *)
		ipSrcContainer2	:	ITcVnContainer;	(* Source container 2 *)
		ipDestContainer	:	REFERENCE TO ITcVnContainer;	(* Returns the resulting container *)
		hrPrev	:	HRESULT;	(* HRESULT indicating the result of previous operations (If SUCCEEDED(hrPrev) equals false, no operation is executed.) *)
	END_VAR

END_FUNCTION

// Functions/Algebraic Image Operations/F_VN_AddImages

	{attribute 'TcIecLibraryType'}
	{attribute 'external_name' := 'F_VN_AddImages_GUID_F4A5C102_2B98_2A50_7D89_ED85590ADDFF'}
	(* Element-wise addition of two images using saturation arithmetics. *)
	FUNCTION F_VN_AddImages : HRESULT
	VAR_INPUT
		ipSrcImage1	:	ITcVnImage;	(* First source image *)
		ipSrcImage2	:	ITcVnImage;	(* Second source image *)
		ipDestImage	:	REFERENCE TO ITcVnImage;	(* Destination image (An appropriate destination image will be created if required.) *)
		hrPrev	:	HRESULT;	(* HRESULT indicating the result of previous operations (If SUCCEEDED(hrPrev) equals false, no operation is executed.) *)
	END_VAR

END_FUNCTION

// Functions/Algebraic Image Operations/F_VN_AddImagesWeighted

	{attribute 'TcIecLibraryType'}
	{attribute 'external_name' := 'F_VN_AddImagesWeighted_GUID_F83539D2_97ED_2044_7403_85A2F59565AF'}
	(* Weighted, element-wise addition of two images using saturation arithmetics. *)
	FUNCTION F_VN_AddImagesWeighted : HRESULT
	VAR_INPUT
		ipSrcImage1	:	ITcVnImage;	(* First source image *)
		ipSrcImage2	:	ITcVnImage;	(* Second source image *)
		ipDestImage	:	REFERENCE TO ITcVnImage;	(* Destination image (An appropriate destination image will be created if required.) *)
		fWeight1	:	LREAL;	(* Weight factor applied to ipSrcImage1 *)
		fWeight2	:	LREAL;	(* Weight factor applied to ipSrcImage2 *)
		fDelta	:	LREAL;	(* Value added to the weighted sum of both images *)
		hrPrev	:	HRESULT;	(* HRESULT indicating the result of previous operations (If SUCCEEDED(hrPrev) equals false, no operation is executed.) *)
	END_VAR

END_FUNCTION

// Functions/Algebraic Image Operations/F_VN_AddImagesWeightedExp

	{attribute 'TcIecLibraryType'}
	{attribute 'external_name' := 'F_VN_AddImagesWeightedExp_GUID_24F170DC_613E_2367_4AA8_2722D0B29B6C'}
	(* Weighted, element-wise addition of two images using saturation arithmetics. *)
	FUNCTION F_VN_AddImagesWeightedExp : HRESULT
	VAR_INPUT
		ipSrcImage1	:	ITcVnImage;	(* First source image *)
		ipSrcImage2	:	ITcVnImage;	(* Second source image *)
		ipDestImage	:	REFERENCE TO ITcVnImage;	(* Destination image (An appropriate destination image will be created if required.) *)
		fWeight1	:	LREAL;	(* Weight factor applied to ipSrcImage1 *)
		fWeight2	:	LREAL;	(* Weight factor applied to ipSrcImage2 *)
		fDelta	:	LREAL;	(* Value added to the weighted sum of both images *)
		eDestType	:	ETcVnElementType;	(* Destination image depth *)
		hrPrev	:	HRESULT;	(* HRESULT indicating the result of previous operations (If SUCCEEDED(hrPrev) equals false, no operation is executed.) *)
	END_VAR

END_FUNCTION

// Functions/Algebraic Image Operations/F_VN_AddScalarToImage

	{attribute 'TcIecLibraryType'}
	{attribute 'external_name' := 'F_VN_AddScalarToImage_GUID_D8601E73_616A_2A97_6934_FADAA36524D3'}
	(* Add a scalar value to each image pixel using saturation arithmetics. *)
	FUNCTION F_VN_AddScalarToImage : HRESULT
	VAR_INPUT
		fScalar	:	LREAL;	(* Scalar value *)
		ipSrcImage	:	ITcVnImage;	(* Source image *)
		ipDestImage	:	REFERENCE TO ITcVnImage;	(* Destination image (An appropriate destination image will be created if required.) *)
		hrPrev	:	HRESULT;	(* HRESULT indicating the result of previous operations (If SUCCEEDED(hrPrev) equals false, no operation is executed.) *)
	END_VAR

END_FUNCTION

// Functions/Algebraic Image Operations/F_VN_AddVectorToImage

	{attribute 'TcIecLibraryType'}
	{attribute 'external_name' := 'F_VN_AddVectorToImage_GUID_4D173667_A863_2F55_6AF5_0775B6B98F51'}
	(* Add a vector (1 element for each image channel) to each image pixel using saturation arithmetics. *)
	FUNCTION F_VN_AddVectorToImage : HRESULT
	VAR_IN_OUT
		aVector	:	TcVnVector4_LREAL;	(* 4-element vector (1 element for each image channel. If the image has less channels, the further vector elements are ignored.) *)
	END_VAR
	VAR_INPUT
		ipSrcImage	:	ITcVnImage;	(* Source image *)
		ipDestImage	:	REFERENCE TO ITcVnImage;	(* Destination image (An appropriate destination image will be created if required.) *)
		hrPrev	:	HRESULT;	(* HRESULT indicating the result of previous operations (If SUCCEEDED(hrPrev) equals false, no operation is executed.) *)
	END_VAR

END_FUNCTION

// Functions/Algebraic Image Operations/F_VN_BitwiseAndImages

	{attribute 'TcIecLibraryType'}
	{attribute 'external_name' := 'F_VN_BitwiseAndImages_GUID_2EBC853A_7DAC_21E7_7613_A230B94A7410'}
	(* Element-wise application of a bit-wise AND operator to two images. *)
	FUNCTION F_VN_BitwiseAndImages : HRESULT
	VAR_INPUT
		ipSrcImage1	:	ITcVnImage;	(* First source image *)
		ipSrcImage2	:	ITcVnImage;	(* Second source image *)
		ipDestImage	:	REFERENCE TO ITcVnImage;	(* Destination image (An appropriate destination image will be created if required.) *)
		hrPrev	:	HRESULT;	(* HRESULT indicating the result of previous operations (If SUCCEEDED(hrPrev) equals false, no operation is executed.) *)
	END_VAR

END_FUNCTION

// Functions/Algebraic Image Operations/F_VN_BitwiseAndImagesExp

	{attribute 'TcIecLibraryType'}
	{attribute 'external_name' := 'F_VN_BitwiseAndImagesExp_GUID_B8463F0A_47B8_22EF_43DF_A7E5C9FA83F7'}
	(* Element-wise application of a bit-wise AND operator to two images. (expert function) *)
	FUNCTION F_VN_BitwiseAndImagesExp : HRESULT
	VAR_INPUT
		ipSrcImage1	:	ITcVnImage;	(* First source image *)
		ipSrcImage2	:	ITcVnImage;	(* Second source image *)
		ipDestImage	:	REFERENCE TO ITcVnImage;	(* Destination image (An appropriate destination image will be created if required.) *)
		ipMask	:	ITcVnImage;	(* Mask to limit the operation to specific pixel positions (mask value 0: skip pixel, mask value > 0: apply operation to pixel) *)
		hrPrev	:	HRESULT;	(* HRESULT indicating the result of previous operations (If SUCCEEDED(hrPrev) equals false, no operation is executed.) *)
	END_VAR

END_FUNCTION

// Functions/Algebraic Image Operations/F_VN_BitwiseAndScalarWithImage

	{attribute 'TcIecLibraryType'}
	{attribute 'external_name' := 'F_VN_BitwiseAndScalarWithImage_GUID_A8309266_56C1_2EA9_65BC_A73F2AF44DB8'}
	(* Bitwise and a scalar value with each image pixel. *)
	FUNCTION F_VN_BitwiseAndScalarWithImage : HRESULT
	VAR_INPUT
		fScalar	:	LREAL;	(* Scalar value *)
		ipSrcImage	:	ITcVnImage;	(* Source image *)
		ipDestImage	:	REFERENCE TO ITcVnImage;	(* Destination image (An appropriate destination image will be created if required.) *)
		hrPrev	:	HRESULT;	(* HRESULT indicating the result of previous operations (If SUCCEEDED(hrPrev) equals false, no operation is executed.) *)
	END_VAR

END_FUNCTION

// Functions/Algebraic Image Operations/F_VN_BitwiseAndVectorWithImage

	{attribute 'TcIecLibraryType'}
	{attribute 'external_name' := 'F_VN_BitwiseAndVectorWithImage_GUID_ACFCD923_EBFB_2782_5A58_E52684A06541'}
	(* Bitwise and a vector (1 element for each image channel) with each image pixel. *)
	FUNCTION F_VN_BitwiseAndVectorWithImage : HRESULT
	VAR_IN_OUT
		aVector	:	TcVnVector4_LREAL;	(* 4-element vector (1 element for each image channel. If the image has less channels, the further vector elements are ignored.) *)
	END_VAR
	VAR_INPUT
		ipSrcImage	:	ITcVnImage;	(* Source image *)
		ipDestImage	:	REFERENCE TO ITcVnImage;	(* Destination image (An appropriate destination image will be created if required.) *)
		hrPrev	:	HRESULT;	(* HRESULT indicating the result of previous operations (If SUCCEEDED(hrPrev) equals false, no operation is executed.) *)
	END_VAR

END_FUNCTION

// Functions/Algebraic Image Operations/F_VN_BitwiseNotImage

	{attribute 'TcIecLibraryType'}
	{attribute 'external_name' := 'F_VN_BitwiseNotImage_GUID_940AB3AD_D0A1_2C97_7396_63D9FD7C9BA5'}
	(* Element-wise application of a bit-wise NOT operator to an image. *)
	FUNCTION F_VN_BitwiseNotImage : HRESULT
	VAR_INPUT
		ipSrcImage	:	ITcVnImage;	(* Source image *)
		ipDestImage	:	REFERENCE TO ITcVnImage;	(* Destination image (An appropriate destination image will be created if required.) *)
		hrPrev	:	HRESULT;	(* HRESULT indicating the result of previous operations (If SUCCEEDED(hrPrev) equals false, no operation is executed.) *)
	END_VAR

END_FUNCTION

// Functions/Algebraic Image Operations/F_VN_BitwiseNotImageExp

	{attribute 'TcIecLibraryType'}
	{attribute 'external_name' := 'F_VN_BitwiseNotImageExp_GUID_AA755875_AE9D_2305_4619_F8FAA2B13236'}
	(* Element-wise application of a bit-wise NOT operator to an image. (expert function) *)
	FUNCTION F_VN_BitwiseNotImageExp : HRESULT
	VAR_INPUT
		ipSrcImage	:	ITcVnImage;	(* Source image *)
		ipDestImage	:	REFERENCE TO ITcVnImage;	(* Destination image (An appropriate destination image will be created if required.) *)
		ipMask	:	ITcVnImage;	(* Mask to limit the operation to specific pixel positions (mask value 0: skip pixel, mask value > 0: apply operation to pixel) *)
		hrPrev	:	HRESULT;	(* HRESULT indicating the result of previous operations (If SUCCEEDED(hrPrev) equals false, no operation is executed.) *)
	END_VAR

END_FUNCTION

// Functions/Algebraic Image Operations/F_VN_BitwiseOrImages

	{attribute 'TcIecLibraryType'}
	{attribute 'external_name' := 'F_VN_BitwiseOrImages_GUID_59A78A1E_30B4_2EF3_572D_1D302EEF9761'}
	(* Element-wise application of a bit-wise OR operator to two images. *)
	FUNCTION F_VN_BitwiseOrImages : HRESULT
	VAR_INPUT
		ipSrcImage1	:	ITcVnImage;	(* First source image *)
		ipSrcImage2	:	ITcVnImage;	(* Second source image *)
		ipDestImage	:	REFERENCE TO ITcVnImage;	(* Destination image (An appropriate destination image will be created if required.) *)
		hrPrev	:	HRESULT;	(* HRESULT indicating the result of previous operations (If SUCCEEDED(hrPrev) equals false, no operation is executed.) *)
	END_VAR

END_FUNCTION

// Functions/Algebraic Image Operations/F_VN_BitwiseOrImagesExp

	{attribute 'TcIecLibraryType'}
	{attribute 'external_name' := 'F_VN_BitwiseOrImagesExp_GUID_F5E964F1_B647_224A_5C0B_EA9F1357C76C'}
	(* Element-wise application of a bit-wise OR operator to two images. (expert function) *)
	FUNCTION F_VN_BitwiseOrImagesExp : HRESULT
	VAR_INPUT
		ipSrcImage1	:	ITcVnImage;	(* First source image *)
		ipSrcImage2	:	ITcVnImage;	(* Second source image *)
		ipDestImage	:	REFERENCE TO ITcVnImage;	(* Destination image (An appropriate destination image will be created if required.) *)
		ipMask	:	ITcVnImage;	(* Mask to limit the operation to specific pixel positions (mask value 0: skip pixel, mask value > 0: apply operation to pixel) *)
		hrPrev	:	HRESULT;	(* HRESULT indicating the result of previous operations (If SUCCEEDED(hrPrev) equals false, no operation is executed.) *)
	END_VAR

END_FUNCTION

// Functions/Algebraic Image Operations/F_VN_BitwiseOrScalarWithImage

	{attribute 'TcIecLibraryType'}
	{attribute 'external_name' := 'F_VN_BitwiseOrScalarWithImage_GUID_9F220629_BF50_2DE4_4037_A931094C40EB'}
	(* Bitwise or a scalar value with each image pixel. *)
	FUNCTION F_VN_BitwiseOrScalarWithImage : HRESULT
	VAR_INPUT
		fScalar	:	LREAL;	(* Scalar value *)
		ipSrcImage	:	ITcVnImage;	(* Source image *)
		ipDestImage	:	REFERENCE TO ITcVnImage;	(* Destination image (An appropriate destination image will be created if required.) *)
		hrPrev	:	HRESULT;	(* HRESULT indicating the result of previous operations (If SUCCEEDED(hrPrev) equals false, no operation is executed.) *)
	END_VAR

END_FUNCTION

// Functions/Algebraic Image Operations/F_VN_BitwiseOrVectorWithImage

	{attribute 'TcIecLibraryType'}
	{attribute 'external_name' := 'F_VN_BitwiseOrVectorWithImage_GUID_D8FA8320_65CA_20B8_62C9_35A8F962C54E'}
	(* Bitwise or a vector (1 element for each image channel) with each image pixel. *)
	FUNCTION F_VN_BitwiseOrVectorWithImage : HRESULT
	VAR_IN_OUT
		aVector	:	TcVnVector4_LREAL;	(* 4-element vector (1 element for each image channel. If the image has less channels, the further vector elements are ignored.) *)
	END_VAR
	VAR_INPUT
		ipSrcImage	:	ITcVnImage;	(* Source image *)
		ipDestImage	:	REFERENCE TO ITcVnImage;	(* Destination image (An appropriate destination image will be created if required.) *)
		hrPrev	:	HRESULT;	(* HRESULT indicating the result of previous operations (If SUCCEEDED(hrPrev) equals false, no operation is executed.) *)
	END_VAR

END_FUNCTION

// Functions/Algebraic Image Operations/F_VN_BitwiseXorImages

	{attribute 'TcIecLibraryType'}
	{attribute 'external_name' := 'F_VN_BitwiseXorImages_GUID_981F8C54_C2B6_2E87_5D2E_394AF0BCBCB4'}
	(* Element-wise application of a bit-wise XOR operator to two images. *)
	FUNCTION F_VN_BitwiseXorImages : HRESULT
	VAR_INPUT
		ipSrcImage1	:	ITcVnImage;	(* First source image *)
		ipSrcImage2	:	ITcVnImage;	(* Second source image *)
		ipDestImage	:	REFERENCE TO ITcVnImage;	(* Destination image (An appropriate destination image will be created if required.) *)
		hrPrev	:	HRESULT;	(* HRESULT indicating the result of previous operations (If SUCCEEDED(hrPrev) equals false, no operation is executed.) *)
	END_VAR

END_FUNCTION

// Functions/Algebraic Image Operations/F_VN_BitwiseXorImagesExp

	{attribute 'TcIecLibraryType'}
	{attribute 'external_name' := 'F_VN_BitwiseXorImagesExp_GUID_CB5E22AE_83BF_2893_68CD_537F9E760265'}
	(* Element-wise application of a bit-wise XOR operator to two images. (expert function) *)
	FUNCTION F_VN_BitwiseXorImagesExp : HRESULT
	VAR_INPUT
		ipSrcImage1	:	ITcVnImage;	(* First source image *)
		ipSrcImage2	:	ITcVnImage;	(* Second source image *)
		ipDestImage	:	REFERENCE TO ITcVnImage;	(* Destination image (An appropriate destination image will be created if required.) *)
		ipMask	:	ITcVnImage;	(* Mask to limit the operation to specific pixel positions (mask value 0: skip pixel, mask value > 0: apply operation to pixel) *)
		hrPrev	:	HRESULT;	(* HRESULT indicating the result of previous operations (If SUCCEEDED(hrPrev) equals false, no operation is executed.) *)
	END_VAR

END_FUNCTION

// Functions/Algebraic Image Operations/F_VN_BitwiseXorScalarWithImage

	{attribute 'TcIecLibraryType'}
	{attribute 'external_name' := 'F_VN_BitwiseXorScalarWithImage_GUID_A1DBCBC0_5922_29F4_7AC7_980DDF7B540A'}
	(* Bitwise xor a scalar value with each image pixel. *)
	FUNCTION F_VN_BitwiseXorScalarWithImage : HRESULT
	VAR_INPUT
		fScalar	:	LREAL;	(* Scalar value *)
		ipSrcImage	:	ITcVnImage;	(* Source image *)
		ipDestImage	:	REFERENCE TO ITcVnImage;	(* Destination image (An appropriate destination image will be created if required.) *)
		hrPrev	:	HRESULT;	(* HRESULT indicating the result of previous operations (If SUCCEEDED(hrPrev) equals false, no operation is executed.) *)
	END_VAR

END_FUNCTION

// Functions/Algebraic Image Operations/F_VN_BitwiseXorVectorWithImage

	{attribute 'TcIecLibraryType'}
	{attribute 'external_name' := 'F_VN_BitwiseXorVectorWithImage_GUID_27AD762A_D425_2968_7E8D_9EC26B79E82D'}
	(* Bitwise xor a vector (1 element for each image channel) with each image pixel. *)
	FUNCTION F_VN_BitwiseXorVectorWithImage : HRESULT
	VAR_IN_OUT
		aVector	:	TcVnVector4_LREAL;	(* 4-element vector (1 element for each image channel. If the image has less channels, the further vector elements are ignored.) *)
	END_VAR
	VAR_INPUT
		ipSrcImage	:	ITcVnImage;	(* Source image *)
		ipDestImage	:	REFERENCE TO ITcVnImage;	(* Destination image (An appropriate destination image will be created if required.) *)
		hrPrev	:	HRESULT;	(* HRESULT indicating the result of previous operations (If SUCCEEDED(hrPrev) equals false, no operation is executed.) *)
	END_VAR

END_FUNCTION

// Functions/Algebraic Image Operations/F_VN_BlendImages

	{attribute 'TcIecLibraryType'}
	{attribute 'external_name' := 'F_VN_BlendImages_GUID_4955603C_5515_29FC_43A2_1A469764C83D'}
	(* Blends two images, i.e. dest = (src1 * weight1 + src2 * weight2) / (weight1 + weight2). *)
	FUNCTION F_VN_BlendImages : HRESULT
	VAR_INPUT
		ipSrcImage1	:	ITcVnImage;	(* First source image (ET_USINT or ET_REAL) *)
		ipSrcImage2	:	ITcVnImage;	(* Second source image (same type and size as ipSrcImage1) *)
		ipWeights1	:	ITcVnImage;	(* Weights for ipSrcImage1 (1 channel, ET_REAL) *)
		ipWeights2	:	ITcVnImage;	(* Weights for ipSrcImage2 (1 channel, ET_REAL) *)
		ipDestImage	:	REFERENCE TO ITcVnImage;	(* Destination image (An appropriate destination image will be created if required.) *)
		hrPrev	:	HRESULT;	(* HRESULT indicating the result of previous operations (If SUCCEEDED(hrPrev) equals false, no operation is executed.) *)
	END_VAR

END_FUNCTION

// Functions/Algebraic Image Operations/F_VN_DivideImageByScalar

	{attribute 'TcIecLibraryType'}
	{attribute 'external_name' := 'F_VN_DivideImageByScalar_GUID_88175D24_A650_2612_49CE_A76F5BF67CE3'}
	(* Divide each image pixel by a scalar value using saturation arithmetics. *)
	FUNCTION F_VN_DivideImageByScalar : HRESULT
	VAR_INPUT
		ipSrcImage	:	ITcVnImage;	(* Source image *)
		fScalar	:	LREAL;	(* Scalar value *)
		ipDestImage	:	REFERENCE TO ITcVnImage;	(* Destination image (An appropriate destination image will be created if required.) *)
		hrPrev	:	HRESULT;	(* HRESULT indicating the result of previous operations (If SUCCEEDED(hrPrev) equals false, no operation is executed.) *)
	END_VAR

END_FUNCTION

// Functions/Algebraic Image Operations/F_VN_DivideImageByVector

	{attribute 'TcIecLibraryType'}
	{attribute 'external_name' := 'F_VN_DivideImageByVector_GUID_78E8A3B7_D6D6_2BA4_4B13_64A4B61543AB'}
	(* Divides each image pixel by a vector (1 element for each image channel) using saturation arithmetics. *)
	FUNCTION F_VN_DivideImageByVector : HRESULT
	VAR_INPUT
		ipSrcImage	:	ITcVnImage;	(* Source image *)
	END_VAR
	VAR_IN_OUT
		aVector	:	TcVnVector4_LREAL;	(* 4-element vector (1 element for each image channel. If the image has less channels, the further vector elements are ignored.) *)
	END_VAR
	VAR_INPUT
		ipDestImage	:	REFERENCE TO ITcVnImage;	(* Destination image (An appropriate destination image will be created if required.) *)
		hrPrev	:	HRESULT;	(* HRESULT indicating the result of previous operations (If SUCCEEDED(hrPrev) equals false, no operation is executed.) *)
	END_VAR

END_FUNCTION

// Functions/Algebraic Image Operations/F_VN_DivideImages

	{attribute 'TcIecLibraryType'}
	{attribute 'external_name' := 'F_VN_DivideImages_GUID_981C011C_5C95_2F27_46CC_1E0C64668695'}
	(* Element-wise division of two images using saturation arithmetics. (A division by zero equals zero.) *)
	FUNCTION F_VN_DivideImages : HRESULT
	VAR_INPUT
		ipSrcImage1	:	ITcVnImage;	(* First source image (dividend) *)
		ipSrcImage2	:	ITcVnImage;	(* Second source image (divisor) *)
		ipDestImage	:	REFERENCE TO ITcVnImage;	(* Destination image (An appropriate destination image will be created if required.) *)
		hrPrev	:	HRESULT;	(* HRESULT indicating the result of previous operations (If SUCCEEDED(hrPrev) equals false, no operation is executed.) *)
	END_VAR

END_FUNCTION

// Functions/Algebraic Image Operations/F_VN_DivideScalarByImage

	{attribute 'TcIecLibraryType'}
	{attribute 'external_name' := 'F_VN_DivideScalarByImage_GUID_CB693D21_9286_23F7_7B64_6D2B50B49CC2'}
	(* Divides a scalar value by each image pixel using saturation arithmetics. *)
	FUNCTION F_VN_DivideScalarByImage : HRESULT
	VAR_INPUT
		fScalar	:	LREAL;	(* Scalar value *)
		ipSrcImage	:	ITcVnImage;	(* Source image *)
		ipDestImage	:	REFERENCE TO ITcVnImage;	(* Destination image (An appropriate destination image will be created if required.) *)
		hrPrev	:	HRESULT;	(* HRESULT indicating the result of previous operations (If SUCCEEDED(hrPrev) equals false, no operation is executed.) *)
	END_VAR

END_FUNCTION

// Functions/Algebraic Image Operations/F_VN_DivideVectorByImage

	{attribute 'TcIecLibraryType'}
	{attribute 'external_name' := 'F_VN_DivideVectorByImage_GUID_C04C5E4C_A448_27F1_4B29_2B3AEF84415A'}
	(* Divides a vector (1 element for each image channel) by each image pixel using saturation arithmetics. *)
	FUNCTION F_VN_DivideVectorByImage : HRESULT
	VAR_IN_OUT
		aVector	:	TcVnVector4_LREAL;	(* 4-element vector (1 element for each image channel. If the image has less channels, the further vector elements are ignored.) *)
	END_VAR
	VAR_INPUT
		ipSrcImage	:	ITcVnImage;	(* Source image *)
		ipDestImage	:	REFERENCE TO ITcVnImage;	(* Destination image (An appropriate destination image will be created if required.) *)
		hrPrev	:	HRESULT;	(* HRESULT indicating the result of previous operations (If SUCCEEDED(hrPrev) equals false, no operation is executed.) *)
	END_VAR

END_FUNCTION

// Functions/Algebraic Image Operations/F_VN_ElementwiseExp

	{attribute 'TcIecLibraryType'}
	{attribute 'external_name' := 'F_VN_ElementwiseExp_GUID_E2A78456_BAE7_2722_4DE8_C0EC54E13C43'}
	(* Computes the natural exponent of each pixel value. *)
	FUNCTION F_VN_ElementwiseExp : HRESULT
	VAR_INPUT
		ipSrcImage	:	ITcVnImage;	(* Source image (REAL or LREAL) *)
		ipDestImage	:	REFERENCE TO ITcVnImage;	(* Destination image (Same type and size as ipSrcImage, an appropriate image will be created if required.) *)
		hrPrev	:	HRESULT;	(* HRESULT indicating the result of previous operations (If SUCCEEDED(hrPrev) equals false, no operation is executed.) *)
	END_VAR

END_FUNCTION

// Functions/Algebraic Image Operations/F_VN_ElementwiseLog

	{attribute 'TcIecLibraryType'}
	{attribute 'external_name' := 'F_VN_ElementwiseLog_GUID_FA709E6F_1848_213C_745C_0D86280A7E0A'}
	(* Computes the natural logarithm of each pixel value. *)
	FUNCTION F_VN_ElementwiseLog : HRESULT
	VAR_INPUT
		ipSrcImage	:	ITcVnImage;	(* Source image (REAL or LREAL) *)
		ipDestImage	:	REFERENCE TO ITcVnImage;	(* Destination image (Same type and size as ipSrcImage, an appropriate image will be created if required.) *)
		hrPrev	:	HRESULT;	(* HRESULT indicating the result of previous operations (If SUCCEEDED(hrPrev) equals false, no operation is executed.) *)
	END_VAR

END_FUNCTION

// Functions/Algebraic Image Operations/F_VN_MaxImage

	{attribute 'TcIecLibraryType'}
	{attribute 'external_name' := 'F_VN_MaxImage_GUID_9A391B0F_4653_25C8_77F5_0FAFD9DD106F'}
	(* Element-wise maximum of two images. *)
	FUNCTION F_VN_MaxImage : HRESULT
	VAR_INPUT
		ipSrcImage1	:	ITcVnImage;	(* First source image *)
		ipSrcImage2	:	ITcVnImage;	(* Second source image *)
		ipDestImage	:	REFERENCE TO ITcVnImage;	(* Destination image (An appropriate destination image will be created if required.) *)
		hrPrev	:	HRESULT;	(* HRESULT indicating the result of previous operations (If SUCCEEDED(hrPrev) equals false, no operation is executed.) *)
	END_VAR

END_FUNCTION

// Functions/Algebraic Image Operations/F_VN_MaxImageExp

	{attribute 'TcIecLibraryType'}
	{attribute 'external_name' := 'F_VN_MaxImageExp_GUID_94748E12_8C62_2E0A_5030_A1FE318920B7'}
	(* Element-wise maximum of two images. (expert function) *)
	FUNCTION F_VN_MaxImageExp : HRESULT
	VAR_INPUT
		ipSrcImage1	:	ITcVnImage;	(* First source image *)
		ipSrcImage2	:	ITcVnImage;	(* Second source image *)
		ipDestImage	:	REFERENCE TO ITcVnImage;	(* Destination image (An appropriate destination image will be created if required.) *)
		ipMask	:	ITcVnImage;	(* Mask of type USINT *)
		hrPrev	:	HRESULT;	(* HRESULT indicating the result of previous operations (If SUCCEEDED(hrPrev) equals false, no operation is executed.) *)
	END_VAR

END_FUNCTION

// Functions/Algebraic Image Operations/F_VN_MaxImageWithScalar

	{attribute 'TcIecLibraryType'}
	{attribute 'external_name' := 'F_VN_MaxImageWithScalar_GUID_CFF96FF8_E479_29BD_4172_750138A98CBB'}
	(* Element-wise maximum of image and scalar value. *)
	FUNCTION F_VN_MaxImageWithScalar : HRESULT
	VAR_INPUT
		fScalar	:	LREAL;	(* Scalar value *)
		ipSrcImage	:	ITcVnImage;	(* Source image *)
		ipDestImage	:	REFERENCE TO ITcVnImage;	(* Destination image (An appropriate destination image will be created if required.) *)
		hrPrev	:	HRESULT;	(* HRESULT indicating the result of previous operations (If SUCCEEDED(hrPrev) equals false, no operation is executed.) *)
	END_VAR

END_FUNCTION

// Functions/Algebraic Image Operations/F_VN_MaxImageWithScalarExp

	{attribute 'TcIecLibraryType'}
	{attribute 'external_name' := 'F_VN_MaxImageWithScalarExp_GUID_BFCAC435_0BFB_277D_471A_FC14852E6529'}
	(* Element-wise maximum of image and scalar value. (expert function) *)
	FUNCTION F_VN_MaxImageWithScalarExp : HRESULT
	VAR_INPUT
		fScalar	:	LREAL;	(* Scalar value *)
		ipSrcImage	:	ITcVnImage;	(* Source image *)
		ipDestImage	:	REFERENCE TO ITcVnImage;	(* Destination image (An appropriate destination image will be created if required.) *)
		ipMask	:	ITcVnImage;	(* Mask of type USINT *)
		hrPrev	:	HRESULT;	(* HRESULT indicating the result of previous operations (If SUCCEEDED(hrPrev) equals false, no operation is executed.) *)
	END_VAR

END_FUNCTION

// Functions/Algebraic Image Operations/F_VN_MaxImageWithVector

	{attribute 'TcIecLibraryType'}
	{attribute 'external_name' := 'F_VN_MaxImageWithVector_GUID_2D88E0F7_37A5_2EFF_59D0_C2D18366C6D8'}
	(* Element-wise maximum of image and vector (1 element for each image channel). *)
	FUNCTION F_VN_MaxImageWithVector : HRESULT
	VAR_IN_OUT
		aVector	:	TcVnVector4_LREAL;	(* 4-element vector (1 element for each image channel. If the image has less channels, the further vector elements are ignored.) *)
	END_VAR
	VAR_INPUT
		ipSrcImage	:	ITcVnImage;	(* Source image *)
		ipDestImage	:	REFERENCE TO ITcVnImage;	(* Destination image (An appropriate destination image will be created if required.) *)
		hrPrev	:	HRESULT;	(* HRESULT indicating the result of previous operations (If SUCCEEDED(hrPrev) equals false, no operation is executed.) *)
	END_VAR

END_FUNCTION

// Functions/Algebraic Image Operations/F_VN_MaxImageWithVectorExp

	{attribute 'TcIecLibraryType'}
	{attribute 'external_name' := 'F_VN_MaxImageWithVectorExp_GUID_3D658335_A8E5_2495_58A4_0E2FB8F0F117'}
	(* Element-wise maximum of image and vector (1 element for each image channel). (expert function) *)
	FUNCTION F_VN_MaxImageWithVectorExp : HRESULT
	VAR_IN_OUT
		aVector	:	TcVnVector4_LREAL;	(* 4-element vector (1 element for each image channel. If the image has less channels, the further vector elements are ignored.) *)
	END_VAR
	VAR_INPUT
		ipSrcImage	:	ITcVnImage;	(* Source image *)
		ipDestImage	:	REFERENCE TO ITcVnImage;	(* Destination image (An appropriate destination image will be created if required.) *)
		ipMask	:	ITcVnImage;	(* Mask of type USINT *)
		hrPrev	:	HRESULT;	(* HRESULT indicating the result of previous operations (If SUCCEEDED(hrPrev) equals false, no operation is executed.) *)
	END_VAR

END_FUNCTION

// Functions/Algebraic Image Operations/F_VN_MinImage

	{attribute 'TcIecLibraryType'}
	{attribute 'external_name' := 'F_VN_MinImage_GUID_FAA1306B_1B88_2B8C_5CB4_2E17773C3F88'}
	(* Element-wise minimum of two images. *)
	FUNCTION F_VN_MinImage : HRESULT
	VAR_INPUT
		ipSrcImage1	:	ITcVnImage;	(* First source image *)
		ipSrcImage2	:	ITcVnImage;	(* Second source image *)
		ipDestImage	:	REFERENCE TO ITcVnImage;	(* Destination image (An appropriate destination image will be created if required.) *)
		hrPrev	:	HRESULT;	(* HRESULT indicating the result of previous operations (If SUCCEEDED(hrPrev) equals false, no operation is executed.) *)
	END_VAR

END_FUNCTION

// Functions/Algebraic Image Operations/F_VN_MinImageExp

	{attribute 'TcIecLibraryType'}
	{attribute 'external_name' := 'F_VN_MinImageExp_GUID_1E60EB45_6558_2ED0_69FD_5073B083E920'}
	(* Element-wise minimum of two images. (expert function) *)
	FUNCTION F_VN_MinImageExp : HRESULT
	VAR_INPUT
		ipSrcImage1	:	ITcVnImage;	(* First source image *)
		ipSrcImage2	:	ITcVnImage;	(* Second source image *)
		ipDestImage	:	REFERENCE TO ITcVnImage;	(* Destination image (An appropriate destination image will be created if required.) *)
		ipMask	:	ITcVnImage;	(* Mask of type USINT *)
		hrPrev	:	HRESULT;	(* HRESULT indicating the result of previous operations (If SUCCEEDED(hrPrev) equals false, no operation is executed.) *)
	END_VAR

END_FUNCTION

// Functions/Algebraic Image Operations/F_VN_MinImageWithScalar

	{attribute 'TcIecLibraryType'}
	{attribute 'external_name' := 'F_VN_MinImageWithScalar_GUID_1778222B_A987_2D91_745F_35AE1264309D'}
	(* Element-wise minimum of image and scalar value. *)
	FUNCTION F_VN_MinImageWithScalar : HRESULT
	VAR_INPUT
		fScalar	:	LREAL;	(* Scalar value *)
		ipSrcImage	:	ITcVnImage;	(* Source image *)
		ipDestImage	:	REFERENCE TO ITcVnImage;	(* Destination image (An appropriate destination image will be created if required.) *)
		hrPrev	:	HRESULT;	(* HRESULT indicating the result of previous operations (If SUCCEEDED(hrPrev) equals false, no operation is executed.) *)
	END_VAR

END_FUNCTION

// Functions/Algebraic Image Operations/F_VN_MinImageWithScalarExp

	{attribute 'TcIecLibraryType'}
	{attribute 'external_name' := 'F_VN_MinImageWithScalarExp_GUID_D26F2568_211A_21BD_75F5_B28A73405BD8'}
	(* Element-wise minimum of image and scalar value. (expert function) *)
	FUNCTION F_VN_MinImageWithScalarExp : HRESULT
	VAR_INPUT
		fScalar	:	LREAL;	(* Scalar value *)
		ipSrcImage	:	ITcVnImage;	(* Source image *)
		ipDestImage	:	REFERENCE TO ITcVnImage;	(* Destination image (An appropriate destination image will be created if required.) *)
		ipMask	:	ITcVnImage;	(* Mask of type USINT *)
		hrPrev	:	HRESULT;	(* HRESULT indicating the result of previous operations (If SUCCEEDED(hrPrev) equals false, no operation is executed.) *)
	END_VAR

END_FUNCTION

// Functions/Algebraic Image Operations/F_VN_MinImageWithVector

	{attribute 'TcIecLibraryType'}
	{attribute 'external_name' := 'F_VN_MinImageWithVector_GUID_36B5613A_BA21_2824_6200_CE589D54EB47'}
	(* Element-wise minimum of image and vector (1 element for each image channel). *)
	FUNCTION F_VN_MinImageWithVector : HRESULT
	VAR_IN_OUT
		aVector	:	TcVnVector4_LREAL;	(* 4-element vector (1 element for each image channel. If the image has less channels, the further vector elements are ignored.) *)
	END_VAR
	VAR_INPUT
		ipSrcImage	:	ITcVnImage;	(* Source image *)
		ipDestImage	:	REFERENCE TO ITcVnImage;	(* Destination image (An appropriate destination image will be created if required.) *)
		hrPrev	:	HRESULT;	(* HRESULT indicating the result of previous operations (If SUCCEEDED(hrPrev) equals false, no operation is executed.) *)
	END_VAR

END_FUNCTION

// Functions/Algebraic Image Operations/F_VN_MinImageWithVectorExp

	{attribute 'TcIecLibraryType'}
	{attribute 'external_name' := 'F_VN_MinImageWithVectorExp_GUID_99DAE6B3_3DF1_245E_565B_495FD76EE452'}
	(* Element-wise minimum of image and vector (1 element for each image channel). (expert function) *)
	FUNCTION F_VN_MinImageWithVectorExp : HRESULT
	VAR_IN_OUT
		aVector	:	TcVnVector4_LREAL;	(* 4-element vector (1 element for each image channel. If the image has less channels, the further vector elements are ignored.) *)
	END_VAR
	VAR_INPUT
		ipSrcImage	:	ITcVnImage;	(* Source image *)
		ipDestImage	:	REFERENCE TO ITcVnImage;	(* Destination image (An appropriate destination image will be created if required.) *)
		ipMask	:	ITcVnImage;	(* Mask of type USINT *)
		hrPrev	:	HRESULT;	(* HRESULT indicating the result of previous operations (If SUCCEEDED(hrPrev) equals false, no operation is executed.) *)
	END_VAR

END_FUNCTION

// Functions/Algebraic Image Operations/F_VN_MultiplyImages

	{attribute 'TcIecLibraryType'}
	{attribute 'external_name' := 'F_VN_MultiplyImages_GUID_69121572_F951_25F3_5B89_334BFC21E8A7'}
	(* Element-wise multiplication of two images using saturation arithmetics. *)
	FUNCTION F_VN_MultiplyImages : HRESULT
	VAR_INPUT
		ipSrcImage1	:	ITcVnImage;	(* First source image *)
		ipSrcImage2	:	ITcVnImage;	(* Second source image *)
		ipDestImage	:	REFERENCE TO ITcVnImage;	(* Destination image (An appropriate destination image will be created if required.) *)
		hrPrev	:	HRESULT;	(* HRESULT indicating the result of previous operations (If SUCCEEDED(hrPrev) equals false, no operation is executed.) *)
	END_VAR

END_FUNCTION

// Functions/Algebraic Image Operations/F_VN_MultiplyImageWithScalar

	{attribute 'TcIecLibraryType'}
	{attribute 'external_name' := 'F_VN_MultiplyImageWithScalar_GUID_5A936FC1_21F0_2995_470F_1492CD4E21A6'}
	(* Multiply each image pixel by a scalar value using saturation arithmetics. *)
	FUNCTION F_VN_MultiplyImageWithScalar : HRESULT
	VAR_INPUT
		fScalar	:	LREAL;	(* Scalar value *)
		ipSrcImage	:	ITcVnImage;	(* Source image *)
		ipDestImage	:	REFERENCE TO ITcVnImage;	(* Destination image (An appropriate destination image will be created if required.) *)
		hrPrev	:	HRESULT;	(* HRESULT indicating the result of previous operations (If SUCCEEDED(hrPrev) equals false, no operation is executed.) *)
	END_VAR

END_FUNCTION

// Functions/Algebraic Image Operations/F_VN_MultiplyImageWithVector

	{attribute 'TcIecLibraryType'}
	{attribute 'external_name' := 'F_VN_MultiplyImageWithVector_GUID_B1EEE1C7_4FA6_2EC7_707A_954C1236EBFE'}
	(* Multiply each image pixel by a vector (1 element for each image channel) using saturation arithmetics. *)
	FUNCTION F_VN_MultiplyImageWithVector : HRESULT
	VAR_IN_OUT
		aVector	:	TcVnVector4_LREAL;	(* 4-element vector (1 element for each image channel. If the image has less channels, the further vector elements are ignored.) *)
	END_VAR
	VAR_INPUT
		ipSrcImage	:	ITcVnImage;	(* Source image *)
		ipDestImage	:	REFERENCE TO ITcVnImage;	(* Destination image (An appropriate destination image will be created if required.) *)
		hrPrev	:	HRESULT;	(* HRESULT indicating the result of previous operations (If SUCCEEDED(hrPrev) equals false, no operation is executed.) *)
	END_VAR

END_FUNCTION

// Functions/Algebraic Image Operations/F_VN_SubtractImageFromScalar

	{attribute 'TcIecLibraryType'}
	{attribute 'external_name' := 'F_VN_SubtractImageFromScalar_GUID_53126F39_579F_2B2D_7449_349FE7BCCDDD'}
	(* Subtract each image pixel from a scalar value using saturation arithmetics. *)
	FUNCTION F_VN_SubtractImageFromScalar : HRESULT
	VAR_INPUT
		fScalar	:	LREAL;	(* Scalar value *)
		ipSrcImage	:	ITcVnImage;	(* Source image *)
		ipDestImage	:	REFERENCE TO ITcVnImage;	(* Destination image (An appropriate destination image will be created if required.) *)
		hrPrev	:	HRESULT;	(* HRESULT indicating the result of previous operations (If SUCCEEDED(hrPrev) equals false, no operation is executed.) *)
	END_VAR

END_FUNCTION

// Functions/Algebraic Image Operations/F_VN_SubtractImageFromVector

	{attribute 'TcIecLibraryType'}
	{attribute 'external_name' := 'F_VN_SubtractImageFromVector_GUID_FCE93206_B5D9_27D2_653D_E3B316A99818'}
	(* Subtract each image pixel from a vector (1 element for each image channel) using saturation arithmetics. *)
	FUNCTION F_VN_SubtractImageFromVector : HRESULT
	VAR_IN_OUT
		aVector	:	TcVnVector4_LREAL;	(* 4-element vector (1 element for each image channel. If the image has less channels, the further vector elements are ignored.) *)
	END_VAR
	VAR_INPUT
		ipSrcImage	:	ITcVnImage;	(* Source image *)
		ipDestImage	:	REFERENCE TO ITcVnImage;	(* Destination image (An appropriate destination image will be created if required.) *)
		hrPrev	:	HRESULT;	(* HRESULT indicating the result of previous operations (If SUCCEEDED(hrPrev) equals false, no operation is executed.) *)
	END_VAR

END_FUNCTION

// Functions/Algebraic Image Operations/F_VN_SubtractImages

	{attribute 'TcIecLibraryType'}
	{attribute 'external_name' := 'F_VN_SubtractImages_GUID_781364E9_4C64_234F_77E7_7386B1F5DC0B'}
	(* Element-wise subtraction of two images using saturation arithmetics. *)
	FUNCTION F_VN_SubtractImages : HRESULT
	VAR_INPUT
		ipSrcImage1	:	ITcVnImage;	(* First source image (minuend) *)
		ipSrcImage2	:	ITcVnImage;	(* Second source image (subtrahend) *)
		ipDestImage	:	REFERENCE TO ITcVnImage;	(* Destination image (An appropriate destination image will be created if required.) *)
		hrPrev	:	HRESULT;	(* HRESULT indicating the result of previous operations (If SUCCEEDED(hrPrev) equals false, no operation is executed.) *)
	END_VAR

END_FUNCTION

// Functions/Algebraic Image Operations/F_VN_SubtractScalarFromImage

	{attribute 'TcIecLibraryType'}
	{attribute 'external_name' := 'F_VN_SubtractScalarFromImage_GUID_A1CD886E_7AE3_2A03_68A6_E799950392FF'}
	(* Subtract a scalar value from each image pixel using saturation arithmetics. *)
	FUNCTION F_VN_SubtractScalarFromImage : HRESULT
	VAR_INPUT
		ipSrcImage	:	ITcVnImage;	(* Source image *)
		fScalar	:	LREAL;	(* Scalar value *)
		ipDestImage	:	REFERENCE TO ITcVnImage;	(* Destination image (An appropriate destination image will be created if required.) *)
		hrPrev	:	HRESULT;	(* HRESULT indicating the result of previous operations (If SUCCEEDED(hrPrev) equals false, no operation is executed.) *)
	END_VAR

END_FUNCTION

// Functions/Algebraic Image Operations/F_VN_SubtractVectorFromImage

	{attribute 'TcIecLibraryType'}
	{attribute 'external_name' := 'F_VN_SubtractVectorFromImage_GUID_D1FD4042_C4CA_2984_6EE4_A4B503D4A684'}
	(* Subtract a vector (1 element for each image channel) from each image pixel using saturation arithmetics. *)
	FUNCTION F_VN_SubtractVectorFromImage : HRESULT
	VAR_INPUT
		ipSrcImage	:	ITcVnImage;	(* Source image *)
	END_VAR
	VAR_IN_OUT
		aVector	:	TcVnVector4_LREAL;	(* 4-element vector (1 element for each image channel. If the image has less channels, the further vector elements are ignored.) *)
	END_VAR
	VAR_INPUT
		ipDestImage	:	REFERENCE TO ITcVnImage;	(* Destination image (An appropriate destination image will be created if required.) *)
		hrPrev	:	HRESULT;	(* HRESULT indicating the result of previous operations (If SUCCEEDED(hrPrev) equals false, no operation is executed.) *)
	END_VAR

END_FUNCTION

// Functions/Image Analysis/F_VN_CannyEdgeDetection

	{attribute 'TcIecLibraryType'}
	{attribute 'external_name' := 'F_VN_CannyEdgeDetection_GUID_46E939AA_C6C7_2CA7_6CAB_9CC436B47BCA'}
	(* Find edges using the Canny edge detection algorithm. *)
	FUNCTION F_VN_CannyEdgeDetection : HRESULT
	VAR_INPUT
		ipSrcImage	:	ITcVnImage;	(* Source image (elements of type USINT) *)
		ipDestImage	:	REFERENCE TO ITcVnImage;	(* Destination image (elements of type USINT. An appropriate destination image will be created if required.) *)
		fThresholdLow	:	LREAL;	(* Low threshold *)
		fThresholdHigh	:	LREAL;	(* High threshold *)
		hrPrev	:	HRESULT;	(* HRESULT indicating the result of previous operations (If SUCCEEDED(hrPrev) equals false, no operation is executed.) *)
	END_VAR

END_FUNCTION

// Functions/Image Analysis/F_VN_CannyEdgeDetectionExp

	{attribute 'TcIecLibraryType'}
	{attribute 'external_name' := 'F_VN_CannyEdgeDetectionExp_GUID_86B0EC88_3769_29C1_5AB2_4724888DF6A4'}
	(* Find edges using the Canny edge detection algorithm. (expert function) *)
	FUNCTION F_VN_CannyEdgeDetectionExp : HRESULT
	VAR_INPUT
		ipSrcImage	:	ITcVnImage;	(* Source image (elements of type USINT) *)
		ipDestImage	:	REFERENCE TO ITcVnImage;	(* Destination image (elements of type USINT. An appropriate destination image will be created if required.) *)
		fThresholdLow	:	LREAL;	(* Low threshold *)
		fThresholdHigh	:	LREAL;	(* High threshold *)
		nApertureSize	:	UDINT;	(* Aperture size for the Sobel operator (3, 5, 7) *)
		bL2Gradient	:	BOOL;	(* If true, the more accurate (and slower) L2 norm is used instead of the L1 norm *)
		hrPrev	:	HRESULT;	(* HRESULT indicating the result of previous operations (If SUCCEEDED(hrPrev) equals false, no operation is executed.) *)
	END_VAR

END_FUNCTION

// Functions/Image Analysis/F_VN_ConnectedComponents

	{attribute 'TcIecLibraryType'}
	{attribute 'external_name' := 'F_VN_ConnectedComponents_GUID_8823991C_AF7C_22B1_7139_5D1720D180FB'}
	(* Computes the connected components of an image. *)
	FUNCTION F_VN_ConnectedComponents : HRESULT
	VAR_INPUT
		ipSrcImage	:	ITcVnImage;	(* Source image (USINT, 1 channel, binary) *)
		ipLabelImage	:	REFERENCE TO ITcVnImage;	(* Returns the labels for each source image pixel (1 channel, DINT. An appropriate destination image will be created if required.) *)
	END_VAR
	VAR_IN_OUT
		nLabels	:	DINT;	(* Returns the number of labels *)
	END_VAR
	VAR_INPUT
		hrPrev	:	HRESULT;	(* HRESULT indicating the result of previous operations (If SUCCEEDED(hrPrev) equals false, no operation is executed.) *)
	END_VAR

END_FUNCTION

// Functions/Image Analysis/F_VN_ConnectedComponentsExp

	{attribute 'TcIecLibraryType'}
	{attribute 'external_name' := 'F_VN_ConnectedComponentsExp_GUID_50BE3B4D_4163_2001_737F_0A2CC45DA687'}
	(* Computes the connected components of an image. (expert function) *)
	FUNCTION F_VN_ConnectedComponentsExp : HRESULT
	VAR_INPUT
		ipSrcImage	:	ITcVnImage;	(* Source image (USINT, 1 channel, binary) *)
		ipLabelImage	:	REFERENCE TO ITcVnImage;	(* Returns the labels for each source image pixel (1 channel, type depends on eLabelType. An appropriate destination image will be created if required.) *)
	END_VAR
	VAR_IN_OUT
		nLabels	:	DINT;	(* Returns the number of labels *)
	END_VAR
	VAR_INPUT
		eConnectivity	:	ETcVnPixelConnectivity;	(* Selects if 4- or 8-way pixel connectivity should be used *)
		eLabelType	:	ETcVnElementType;	(* Selects the type of ipLabelImage (only UINT or DINT supported) *)
		eAlgorithm	:	ETcVnConnectedComponentsAlgorithm;	(* Selects the applied algorithm *)
		hrPrev	:	HRESULT;	(* HRESULT indicating the result of previous operations (If SUCCEEDED(hrPrev) equals false, no operation is executed.) *)
	END_VAR

END_FUNCTION

// Functions/Image Analysis/F_VN_ConnectedComponentsWithStats

	{attribute 'TcIecLibraryType'}
	{attribute 'external_name' := 'F_VN_ConnectedComponentsWithStats_GUID_E6670130_0B6E_2A52_73C9_6501E9329CF3'}
	(* Computes the connected components and corresponding statistics of an image. *)
	FUNCTION F_VN_ConnectedComponentsWithStats : HRESULT
	VAR_INPUT
		ipSrcImage	:	ITcVnImage;	(* Source image (USINT, 1 channel, binary) *)
		ipLabelImage	:	REFERENCE TO ITcVnImage;	(* Returns the labels for each source image pixel (1 channel, DINT. An appropriate destination image will be created if required.) *)
		ipBoundingBoxes	:	REFERENCE TO ITcVnContainer;	(* Returns the bounding boxes for each labeled region. (ContainerType_Vector_TcVnRectangle_DINT; Non-zero interface pointers are reused.) *)
		ipNumPixels	:	REFERENCE TO ITcVnContainer;	(* Returns the number of pixels for each labeled region. (ContainerType_Vector_DINT; Non-zero interface pointers are reused.) *)
		ipCentroids	:	REFERENCE TO ITcVnContainer;	(* Returns the centroids for each labeled region. (ContainerType_Vector_TcVnPoint2_LREAL; Non-zero interface pointers are reused.) *)
	END_VAR
	VAR_IN_OUT
		nLabels	:	DINT;	(* Returns the number of labels *)
	END_VAR
	VAR_INPUT
		hrPrev	:	HRESULT;	(* HRESULT indicating the result of previous operations (If SUCCEEDED(hrPrev) equals false, no operation is executed.) *)
	END_VAR

END_FUNCTION

// Functions/Image Analysis/F_VN_ConnectedComponentsWithStatsExp

	{attribute 'TcIecLibraryType'}
	{attribute 'external_name' := 'F_VN_ConnectedComponentsWithStatsExp_GUID_2E71A1A6_0A39_24BC_5057_6B43DA203F8B'}
	(* Computes the connected components and corresponding statistics of an image. (expert function) *)
	FUNCTION F_VN_ConnectedComponentsWithStatsExp : HRESULT
	VAR_INPUT
		ipSrcImage	:	ITcVnImage;	(* Source image (USINT, 1 channel, binary) *)
		ipLabelImage	:	REFERENCE TO ITcVnImage;	(* Returns the labels for each source image pixel (1 channel, DINT. An appropriate destination image will be created if required.) *)
		ipBoundingBoxes	:	REFERENCE TO ITcVnContainer;	(* Returns the bounding boxes for each labeled region. (ContainerType_Vector_TcVnRectangle_DINT; Non-zero interface pointers are reused.) *)
		ipNumPixels	:	REFERENCE TO ITcVnContainer;	(* Returns the number of pixels for each labeled region. (ContainerType_Vector_DINT; Non-zero interface pointers are reused.) *)
		ipCentroids	:	REFERENCE TO ITcVnContainer;	(* Returns the centroids for each labeled region. (ContainerType_Vector_TcVnPoint2_LREAL; Non-zero interface pointers are reused.) *)
	END_VAR
	VAR_IN_OUT
		nLabels	:	DINT;	(* Returns the number of labels *)
	END_VAR
	VAR_INPUT
		eConnectivity	:	ETcVnPixelConnectivity;	(* Selects if 4- or 8-way pixel connectivity should be used *)
		eLabelType	:	ETcVnElementType;	(* Selects the type of ipLabelImage (only UINT or DINT supported) *)
		eAlgorithm	:	ETcVnConnectedComponentsAlgorithm;	(* Selects the applied algorithm *)
		hrPrev	:	HRESULT;	(* HRESULT indicating the result of previous operations (If SUCCEEDED(hrPrev) equals false, no operation is executed.) *)
	END_VAR

END_FUNCTION

// Functions/Image Analysis/F_VN_CountNonZeroPixels

	{attribute 'TcIecLibraryType'}
	{attribute 'external_name' := 'F_VN_CountNonZeroPixels_GUID_769F9C03_906B_2846_606F_043D88D9F335'}
	(* Counts the non-zero pixels in a single-channel image (e.g. useful to analyze threshold results). *)
	FUNCTION F_VN_CountNonZeroPixels : HRESULT
	VAR_INPUT
		ipSrcImage	:	ITcVnImage;	(* Source image (1 channel) *)
	END_VAR
	VAR_IN_OUT
		nNonZero	:	ULINT;	(* Returns the number of non-zero pixels in ipSrcImage *)
	END_VAR
	VAR_INPUT
		hrPrev	:	HRESULT;	(* HRESULT indicating the result of previous operations (If SUCCEEDED(hrPrev) equals false, no operation is executed.) *)
	END_VAR

END_FUNCTION

// Functions/Image Analysis/F_VN_DistanceTransformation

	{attribute 'TcIecLibraryType'}
	{attribute 'external_name' := 'F_VN_DistanceTransformation_GUID_A522DFC7_0119_29FC_5B10_BD0439AC25AE'}
	(* Calculates the distance transformation, which is the distance to the closest zero pixel in a binary image. *)
	FUNCTION F_VN_DistanceTransformation : HRESULT
	VAR_INPUT
		ipSrcImage	:	ITcVnImage;	(* Source image (USINT, 1 channel) *)
		ipDestImage	:	REFERENCE TO ITcVnImage;	(* Destination image (REAL, 1 channel. An appropriate destination image will be created if required.) *)
		eDistanceType	:	ETcVnDistanceType;	(* Distance computation method (supported: L1, L2, C) *)
		eMaskSize	:	ETcVnDistanceTransformationMask;	(* Size of the distance transformation mask *)
		hrPrev	:	HRESULT;	(* HRESULT indicating the result of previous operations (If SUCCEEDED(hrPrev) equals false, no operation is executed.) *)
	END_VAR

END_FUNCTION

